query := TOF_Core.GenericValueFactory.FromIntReference(value := keys[2]);
position := _Dictionary.GetKeyPosition(key := keys[2]);
genericPosition := _Dictionary.GetGenericKeyPosition(key := query, releaseKey := FALSE);

Assert.ThatBool(
	actual := position >= 0 AND_THEN position < _Dictionary.Length,
	message := "Key 2 must have a valid current position"
).IsTrue();

Assert.ThatDInt(
	actual := genericPosition,
	message := "Both lookup forms must return the same position for key 2"
).ToBe(expected := position);

FOR i := 0 TO 6 DO
	found := _Dictionary.TryGetValueByKey(key := keys[i], value => value);

	IF i = 3 THEN
		Assert.ThatBool(
			actual := found AND_THEN value.AsString255() = copyReplacement,
			message := "SetCopy must replace the value of key 3"
		).IsTrue();
	ELSIF i = 5 THEN
		Assert.ThatBool(
			actual := found AND_THEN value.AsString255() = _ReplacementValue,
			message := "SetGeneric must replace the value of key 5"
		).IsTrue();
	ELSE
		Assert.ThatBool(
			actual := found AND_THEN value.AsString255() = values[i],
			message := TOF_Core.WideStrings.Concat255("Expected original value at key ", TO_WSTRING(i))
		).IsTrue();
	END_IF
END_FOR

found := _Dictionary.TryGetValueByGenericKey(key := query, releaseKey := FALSE, value => value);

Assert.ThatBool(
	actual := found AND_THEN value.AsString255() = 'String2',
	message := "Generic lookup must return the original value of key 2"
).IsTrue();

position := _Dictionary.GetKeyPosition(key := keys[3]);

IF position < 0 OR_ELSE position >= _Dictionary.Length THEN
	RecordFailure(message := "Updated key 3 must have a valid position");

	RETURN;
END_IF

pair REF= _Dictionary.GetKeyValuePairByIndex(index := position);

Assert.ThatBool(
	actual := __ISVALIDREF(pair) AND_THEN pair.Key.AsInt() = INT#3
		AND_THEN pair.Value.AsString255() = copyReplacement,
	message := "The indexed pair must match both the queried key and its updated value"
).IsTrue();
END_METHOD

(*!
<summary>Clears the fixture before the runner publishes the result.</summary>
<description>
Also runs after an unexpected exception interrupts the case.
</description>
*)
METHOD PROTECTED AfterTest
_Dictionary.Clear();
END_METHOD

//! <summary>Borrows the concrete class name. Callers must not modify it.</summary>
{attribute 'monitoring' := 'call'}
PROPERTY ClassName : REFERENCE TO STRING
GET
ClassName REF= _ClassName;
END_GET
END_PROPERTY

//! <summary>Borrows the compiler-initialized namespace name. Callers must not modify it.</summary>
{attribute 'monitoring' := 'call'}
PROPERTY NamespaceName : REFERENCE TO STRING
GET
NamespaceName REF= CurrentNamespace.Name;
END_GET
END_PROPERTY

//! <summary>Reports the concrete instance size in bytes.</summary>
{attribute 'monitoring' := 'call'}
PROPERTY SelfSize : ULINT
GET
SelfSize := XSIZEOF(THIS^);
END_GET
END_PROPERTY

END_FUNCTION_BLOCK

// ---- Tests/Collections/DictionaryRemoveTest.TcPOU
(*
SPDX-FileCopyrightText: c 2026 Oleksandr Tiutyk <trofimich@gmail.com>
SPDX-License-Identifier: MIT
License: https://opensource.org/license/mit
*)

(*!
<summary>Checks removal by current position and by both key forms.</summary>
<description>
Borrows one group-owned dictionary reserved for this case. Use from one task at a stable address.
Teardown clears entries owned by the dictionary before publication.
</description>
*)

{attribute 'no_assign'}
{attribute 'no_explicit_call' := 'do not call this function block directly'}
FUNCTION_BLOCK DictionaryRemoveTest EXTENDS TOF_Testing.SingleCycleTest
VAR_STAT
	{attribute 'hide'}
	_ClassName : STRING := __POUNAME();
END_VAR
VAR
	_Dictionary : TOF_Collections.IDictionary;
END_VAR

(*!
<summary>Clears the fixture before the runner publishes the result.</summary>
<description>
Also runs after an unexpected exception interrupts the case.
</description>
*)
METHOD PROTECTED AfterTest
_Dictionary.Clear();
END_METHOD

//! <summary>Borrows the concrete class name. Callers must not modify it.</summary>
{attribute 'monitoring' := 'call'}
PROPERTY ClassName : REFERENCE TO STRING
GET
ClassName REF= _ClassName;
END_GET
END_PROPERTY

(*!
<summary>Checks removal by current position and by both key forms.</summary>
*)
METHOD PROTECTED ExecuteTest
VAR
	keys : ARRAY [0..6] OF INT := [0, 1, 2, 3, 4, 5, 6];
	values : ARRAY [0..6] OF STRING :=
		['String0', 'String1', 'String2', 'String3', 'String4', 'String5', 'String6'];
	i : DINT;
	position : DINT;
	query : TOF_Core.GENERIC_VALUE;
	removed : BOOL;
END_VAR
FOR i := 6 TO 0 BY -1 DO
	_Dictionary.SetCopy(key := keys[i], value := values[i]);
END_FOR

_Dictionary.SetCopy(key := keys[3], value := values[3]);

position := _Dictionary.GetKeyPosition(key := keys[3]);

IF position < 0 OR_ELSE position >= _Dictionary.Length THEN
	RecordFailure(message := "Key 3 must have a valid position before removal");

	RETURN;
END_IF

_Dictionary.RemoveAt(index := position);

Assert.ThatBool(
	actual := _Dictionary.Length = 6 AND_THEN NOT _Dictionary.ContainsKey(key := keys[3]),
	message := "RemoveAt must remove only key 3"
).IsTrue();

_Dictionary.TryRemoveByKey(key := keys[2], removed => removed);

Assert.ThatBool(
	actual := removed AND_THEN _Dictionary.Length = 5 AND_THEN NOT _Dictionary.ContainsKey(key := keys[2]),
	message := "TryRemoveByKey must remove key 2 and report success"
).IsTrue();

query := TOF_Core.GenericValueFactory.FromIntReference(value := keys[1]);
_Dictionary.TryRemoveByGenericKey(key := query, releaseKey := FALSE, removed => removed);

Assert.ThatBool(
	actual := removed AND_THEN _Dictionary.Length = 4 AND_THEN NOT _Dictionary.ContainsKey(key := keys[1]),
	message := "TryRemoveByGenericKey must remove key 1 and report success"
).IsTrue();

_Dictionary.TryRemoveByGenericKey(key := query, releaseKey := FALSE, removed => removed);

Assert.ThatBool(
	actual := NOT removed AND_THEN _Dictionary.Length = 4,
	message := "A second removal of key 1 must leave the dictionary unchanged"
).IsTrue();

FOR i := 4 TO 6 DO
	Assert.ThatBool(
		actual := _Dictionary.ContainsKey(key := keys[i]),
		message := TOF_Core.WideStrings.Concat255("Removal must preserve key ", TO_WSTRING(i))
	).IsTrue();
END_FOR

Assert.ThatBool(
	actual := _Dictionary.ContainsKey(key := keys[0]),
	message := "Removal must preserve key 0"
).IsTrue();
END_METHOD

(*!
<summary>Binds the dictionary fixture for this case.</summary>
<description>
Stores a borrowed interface without invoking the fixture. The owning group keeps it alive and
reserves it for this case. TestElement initializes the name and parent.
</description>
<param name="name">Display name of this case.</param>
<param name="parent">Group that owns this case.</param>
<param name="dictionary">Required live dictionary reserved for this case.</param>
*)
METHOD FB_init : BOOL
VAR_INPUT
	bInitRetains: BOOL; // TRUE: the retain variables are initialized (reset warm / reset cold)
	bInCopyCode: BOOL; // TRUE: the instance will be copied to the copy code afterward (online change)
	name : WSTRING;
	parent : TOF_Testing.ITestElement;
	dictionary : TOF_Collections.IDictionary;
END_VAR
_Dictionary := dictionary;
FB_init := TRUE;
END_METHOD

//! <summary>Borrows the compiler-initialized namespace name. Callers must not modify it.</summary>
{attribute 'monitoring' := 'call'}
PROPERTY NamespaceName : REFERENCE TO STRING
GET
NamespaceName REF= CurrentNamespace.Name;
END_GET
END_PROPERTY

//! <summary>Reports the concrete instance size in bytes.</summary>
{attribute 'monitoring' := 'call'}
PROPERTY SelfSize : ULINT
GET
SelfSize := XSIZEOF(THIS^);
END_GET
END_PROPERTY

END_FUNCTION_BLOCK

// ---- Tests/Collections/DictionaryContainsTest.TcPOU
(*
SPDX-FileCopyrightText: c 2026 Oleksandr Tiutyk <trofimich@gmail.com>
SPDX-License-Identifier: MIT
License: https://opensource.org/license/mit
*)

(*!
<summary>Checks matching and missing keys with raw and borrowed generic queries.</summary>
<description>
Borrows one group-owned dictionary reserved for this case. Use from one task at a stable address.
Teardown clears entries owned by the dictionary before publication.
</description>
*)

{attribute 'no_assign'}
{attribute 'no_explicit_call' := 'do not call this function block directly'}
FUNCTION_BLOCK DictionaryContainsTest EXTENDS TOF_Testing.SingleCycleTest
VAR_STAT
	{attribute 'hide'}
	_ClassName : STRING := __POUNAME();
END_VAR
VAR
	_Dictionary : TOF_Collections.IDictionary;
END_VAR

(*!
<summary>Clears the fixture before the runner publishes the result.</summary>
<description>
Also runs after an unexpected exception interrupts the case.
</description>
*)
METHOD PROTECTED AfterTest
_Dictionary.Clear();
END_METHOD

//! <summary>Borrows the concrete class name. Callers must not modify it.</summary>
{attribute 'monitoring' := 'call'}
PROPERTY ClassName : REFERENCE TO STRING
GET
ClassName REF= _ClassName;
END_GET
END_PROPERTY

(*!
<summary>Checks matching and missing keys with raw and borrowed generic queries.</summary>
*)
METHOD PROTECTED ExecuteTest
VAR
	keys : ARRAY [0..6] OF INT := [0, 1, 2, 3, 4, 5, 6];
	values : ARRAY [0..6] OF STRING :=
		['String0', 'String1', 'String2', 'String3', 'String4', 'String5', 'String6'];
	i : DINT;
	missingKey : INT := 9;
	query : TOF_Core.GENERIC_VALUE;
END_VAR
FOR i := 6 TO 0 BY -1 DO
	_Dictionary.SetCopy(key := keys[i], value := values[i]);
END_FOR

_Dictionary.SetCopy(key := keys[3], value := values[3]);

Assert.ThatBool(
	actual := _Dictionary.ContainsKey(key := keys[3]),
	message := "ContainsKey must find the stored key"
).IsTrue();

Assert.ThatBool(
	actual := _Dictionary.ContainsKey(key := missingKey),
	message := "ContainsKey must reject an absent key"
).IsFalse();

query := TOF_Core.GenericValueFactory.FromIntReference(value := keys[3]);
Assert.ThatBool(
	actual := _Dictionary.ContainsGenericKey(key := query, releaseKey := FALSE),
	message := "ContainsGenericKey must find the stored key"
).IsTrue();

query := TOF_Core.GenericValueFactory.FromIntReference(value := missingKey);
Assert.ThatBool(
	actual := _Dictionary.ContainsGenericKey(key := query, releaseKey := FALSE),
	message := "ContainsGenericKey must reject an absent key"
).IsFalse();

Assert.ThatDInt(
	actual := _Dictionary.Length,
	message := "Lookup must preserve all seven entries"
).ToBe(expected := DINT#7);
END_METHOD

(*!
<summary>Binds the dictionary fixture for this case.</summary>
<description>
Stores a borrowed interface without invoking the fixture. The owning group keeps it alive and
reserves it for this case. TestElement initializes the name and parent.
</description>
<param name="name">Display name of this case.</param>
<param name="parent">Group that owns this case.</param>
<param name="dictionary">Required live dictionary reserved for this case.</param>
*)
METHOD FB_init : BOOL
VAR_INPUT
	bInitRetains: BOOL; // TRUE: the retain variables are initialized (reset warm / reset cold)
	bInCopyCode: BOOL; // TRUE: the instance will be copied to the copy code afterward (online change)
	name : WSTRING;
	parent : TOF_Testing.ITestElement;
	dictionary : TOF_Collections.IDictionary;
END_VAR
_Dictionary := dictionary;
FB_init := TRUE;
END_METHOD

//! <summary>Borrows the compiler-initialized namespace name. Callers must not modify it.</summary>
{attribute 'monitoring' := 'call'}
PROPERTY NamespaceName : REFERENCE TO STRING
GET
NamespaceName REF= CurrentNamespace.Name;
END_GET
END_PROPERTY

//! <summary>Reports the concrete instance size in bytes.</summary>
{attribute 'monitoring' := 'call'}
PROPERTY SelfSize : ULINT
GET
SelfSize := XSIZEOF(THIS^);
END_GET
END_PROPERTY

END_FUNCTION_BLOCK

// ---- Tests/Collections/Dynamic/DynamicDictionaryClearTest.TcPOU
(*
SPDX-FileCopyrightText: c 2026 Oleksandr Tiutyk <trofimich@gmail.com>
SPDX-License-Identifier: MIT
License: https://opensource.org/license/mit
*)

(*!
<summary>Checks clearing grown entries and rebuilding a usable index on reuse.</summary>
<description>
Owns a dynamic dictionary and copied pairs at a stable address. Run from one task.
Teardown releases remaining entries and dynamic storage.
</description>
*)

{attribute 'no_assign'}
{attribute 'no_explicit_call' := 'do not call this function block directly'}
FUNCTION_BLOCK DynamicDictionaryClearTest EXTENDS TOF_Testing.SingleCycleTest
VAR_STAT
	{attribute 'hide'}
	_ClassName : STRING := __POUNAME();
END_VAR
VAR
	_Dictionary : TOF_Collections.Dictionary<0>(keyValidator := 0, valueValidator := 0, keyEqualityComparer := 0);
END_VAR

(*!
<summary>Checks clearing grown entries and rebuilding a usable index on reuse.</summary>
*)
METHOD PROTECTED ExecuteTest
VAR
	keys : ARRAY [0..6] OF INT := [0, 1, 2, 3, 4, 5, 6];
	values : ARRAY [0..6] OF STRING :=
		['String0', 'String1', 'String2', 'String3', 'String4', 'String5', 'String6'];
	i : DINT;
	value : TOF_Core.GENERIC_VALUE;
	found : BOOL;
END_VAR
_Dictionary.DefaultDynamicAllocationElementCount := BYTE#2;

FOR i := 6 TO 0 BY -1 DO
	_Dictionary.SetCopy(key := keys[i], value := values[i]);
END_FOR

Assert.ThatBool(
	actual := _Dictionary.Length = 7 AND_THEN _Dictionary.Capacity = 8,
	message := "The clear fixture must start with grown capacity"
).IsTrue();

FOR i := 0 TO 6 DO
	found := _Dictionary.TryGetValueByKey(key := keys[i], value => value);

	Assert.ThatBool(
		actual := found AND_THEN value.AsString255() = values[i],
		message := TOF_Core.WideStrings.Concat255("Growth must preserve the pair at key ", TO_WSTRING(i))
	).IsTrue();
END_FOR

_Dictionary.Clear();

Assert.ThatBool(
	actual := _Dictionary.Empty AND_THEN _Dictionary.Length = 0 AND_THEN _Dictionary.Capacity = 0,
	message := "Clear must empty the dictionary and release capacity"
).IsTrue();

Assert.ThatBool(
	actual := _Dictionary.ContainsKey(key := keys[3]),
	message := "The cleared index must not find an old key"
).IsFalse();

_Dictionary.Clear();
_Dictionary.SetCopy(key := keys[3], value := values[6]);

found := _Dictionary.TryGetValueByKey(key := keys[3], value => value);

Assert.ThatBool(
	actual := found AND_THEN value.AsString255() = 'String6',
	message := "Reinsertion must make the new value visible"
).IsTrue();

Assert.ThatBool(
	actual := _Dictionary.Length = 1 AND_THEN _Dictionary.Capacity = 2,
	message := "Reinsertion must allocate only the initial capacity"
).IsTrue();
END_METHOD

(*!
<summary>Clears the fixture before the runner publishes the result.</summary>
<description>
Also runs after an unexpected exception interrupts the case.
</description>
*)
METHOD PROTECTED AfterTest
_Dictionary.Clear();
END_METHOD

//! <summary>Borrows the concrete class name. Callers must not modify it.</summary>
{attribute 'monitoring' := 'call'}
PROPERTY ClassName : REFERENCE TO STRING
GET
ClassName REF= _ClassName;
END_GET
END_PROPERTY

//! <summary>Borrows the compiler-initialized namespace name. Callers must not modify it.</summary>
{attribute 'monitoring' := 'call'}
PROPERTY NamespaceName : REFERENCE TO STRING
GET
NamespaceName REF= CurrentNamespace.Name;
END_GET
END_PROPERTY

//! <summary>Reports the concrete instance size in bytes.</summary>
{attribute 'monitoring' := 'call'}
PROPERTY SelfSize : ULINT
GET
SelfSize := XSIZEOF(THIS^);
END_GET
END_PROPERTY

END_FUNCTION_BLOCK

// ---- Tests/Collections/Static/StaticDictionaryTestGroup.TcPOU
(*
SPDX-FileCopyrightText: c 2026 Oleksandr Tiutyk <trofimich@gmail.com>
SPDX-License-Identifier: MIT
License: https://opensource.org/license/mit
*)

(*!
<summary>Groups fixed-capacity dictionary lookup, update, removal, clear and overflow cases.</summary>
<description>
Owns the child cases, their fixed registration array and the dictionaries borrowed by the common cases.
Each borrowed fixture is reserved for its case throughout the group lifetime. Use from one task at a stable address.
</description>
*)

{attribute 'no_assign'}
{attribute 'no_explicit_call' := 'do not call this function block directly'}
FUNCTION_BLOCK StaticDictionaryTestGroup EXTENDS TOF_Testing.TestGroup<5>
VAR_STAT
	{attribute 'hide'}
	_ClassName : STRING := __POUNAME();
END_VAR
VAR
	_SetAndGetDictionary : TOF_Collections.Dictionary<7>(keyValidator := 0, valueValidator := 0, keyEqualityComparer := 0);
	_RemoveDictionary : TOF_Collections.Dictionary<7>(keyValidator := 0, valueValidator := 0, keyEqualityComparer := 0);
	_ContainsDictionary : TOF_Collections.Dictionary<7>(keyValidator := 0, valueValidator := 0, keyEqualityComparer := 0);

	_SetAndGet : DictionarySetAndGetTest(name := "SetAndGet", parent := THIS^, dictionary := _SetAndGetDictionary);
	_Remove : DictionaryRemoveTest(name := "Remove", parent := THIS^, dictionary := _RemoveDictionary);
	_Contains : DictionaryContainsTest(name := "Contains", parent := THIS^, dictionary := _ContainsDictionary);
	_Clear : StaticDictionaryClearTest(name := "Clear", parent := THIS^);
	_Overflow : StaticDictionaryOverflowTest(name := "Overflow", parent := THIS^);

	_Children : ARRAY [0.._ChildCount - 1] OF TOF_Testing.ITestElement :=
	[
		_SetAndGet,
		_Remove,
		_Contains,
		_Clear,
		_Overflow
	];
END_VAR

//! <summary>Borrows the fixed child array. Callers must not modify it.</summary>
{attribute 'monitoring' := 'call'}
PROPERTY Children : REFERENCE TO ARRAY [0.._ChildCount - 1] OF TOF_Testing.ITestElement
GET
Children REF= _Children;
END_GET
END_PROPERTY

//! <summary>Borrows the concrete class name. Callers must not modify it.</summary>
{attribute 'monitoring' := 'call'}
PROPERTY ClassName : REFERENCE TO STRING
GET
ClassName REF= _ClassName;
END_GET
END_PROPERTY

//! <summary>Borrows the compiler-initialized namespace name. Callers must not modify it.</summary>
{attribute 'monitoring' := 'call'}
PROPERTY NamespaceName : REFERENCE TO STRING
GET
NamespaceName REF= CurrentNamespace.Name;
END_GET
END_PROPERTY

//! <summary>Reports the concrete instance size in bytes.</summary>
{attribute 'monitoring' := 'call'}
PROPERTY SelfSize : ULINT
GET
SelfSize := XSIZEOF(THIS^);
END_GET
END_PROPERTY

END_FUNCTION_BLOCK

// ---- Tests/Collections/Static/StaticDictionaryClearTest.TcPOU
(*
SPDX-FileCopyrightText: c 2026 Oleksandr Tiutyk <trofimich@gmail.com>
SPDX-License-Identifier: MIT
License: https://opensource.org/license/mit
*)

(*!
<summary>Checks clearing a full inline index and refilling its slots.</summary>
<description>
Owns a fixed-capacity dictionary and copied pairs at a stable address. Run from one task.
Teardown clears surviving entries before publication.
</description>
*)

{attribute 'no_assign'}
{attribute 'no_explicit_call' := 'do not call this function block directly'}
FUNCTION_BLOCK StaticDictionaryClearTest EXTENDS TOF_Testing.SingleCycleTest
VAR_STAT
	{attribute 'hide'}
	_ClassName : STRING := __POUNAME();
END_VAR
VAR
	_Dictionary : TOF_Collections.Dictionary<7>(keyValidator := 0, valueValidator := 0, keyEqualityComparer := 0);
END_VAR

(*!
<summary>Checks clearing a full inline index and refilling its slots.</summary>
*)
METHOD PROTECTED ExecuteTest
VAR
	keys : ARRAY [0..6] OF INT := [0, 1, 2, 3, 4, 5, 6];
	values : ARRAY [0..6] OF STRING :=
		['String0', 'String1', 'String2', 'String3', 'String4', 'String5', 'String6'];
	i : DINT;
	value : TOF_Core.GENERIC_VALUE;
	found : BOOL;
END_VAR
FOR i := 6 TO 0 BY -1 DO
	_Dictionary.SetCopy(key := keys[i], value := values[i]);
END_FOR

Assert.ThatBool(
	actual := _Dictionary.Full AND_THEN _Dictionary.Length = 7,
	message := "The clear fixture must start full"
).IsTrue();

_Dictionary.Clear();

Assert.ThatBool(
	actual := _Dictionary.Empty AND_THEN _Dictionary.Length = 0 AND_THEN NOT _Dictionary.Full,
	message := "Clearing a full dictionary must make every slot available"
).IsTrue();

Assert.ThatDInt(
	actual := _Dictionary.Capacity,
	message := "Clearing must preserve inline capacity"
).ToBe(expected := DINT#7);

FOR i := 0 TO 6 DO
	Assert.ThatBool(
		actual := _Dictionary.ContainsKey(key := keys[i]),
		message := TOF_Core.WideStrings.Concat255("Clear must hide old key ", TO_WSTRING(i))
	).IsFalse();
END_FOR

FOR i := 0 TO 6 DO
	_Dictionary.SetCopy(key := keys[i], value := values[6 - i]);
END_FOR

Assert.ThatBool(
	actual := _Dictionary.Full AND_THEN _Dictionary.Length = 7,
	message := "Refilling must reuse all seven slots"
).IsTrue();

FOR i := 0 TO 6 DO
	found := _Dictionary.TryGetValueByKey(key := keys[i], value => value);

	Assert.ThatBool(
		actual := found AND_THEN value.AsString255() = values[6 - i],
		message := TOF_Core.WideStrings.Concat255("Refill must return the new value at key ", TO_WSTRING(i))
	).IsTrue();
END_FOR
END_METHOD

(*!
<summary>Clears the fixture before the runner publishes the result.</summary>
<description>
Also runs after an unexpected exception interrupts the case.
</description>
*)
METHOD PROTECTED AfterTest
_Dictionary.Clear();
END_METHOD

//! <summary>Borrows the concrete class name. Callers must not modify it.</summary>
{attribute 'monitoring' := 'call'}
PROPERTY ClassName : REFERENCE TO STRING
GET
ClassName REF= _ClassName;
END_GET
END_PROPERTY

//! <summary>Borrows the compiler-initialized namespace name. Callers must not modify it.</summary>
{attribute 'monitoring' := 'call'}
PROPERTY NamespaceName : REFERENCE TO STRING
GET
NamespaceName REF= CurrentNamespace.Name;
END_GET
END_PROPERTY

//! <summary>Reports the concrete instance size in bytes.</summary>
{attribute 'monitoring' := 'call'}
PROPERTY SelfSize : ULINT
GET
SelfSize := XSIZEOF(THIS^);
END_GET
END_PROPERTY

END_FUNCTION_BLOCK

// ---- Tests/Collections/Static/StaticDictionaryOverflowTest.TcPOU
(*
SPDX-FileCopyrightText: c 2026 Oleksandr Tiutyk <trofimich@gmail.com>
SPDX-License-Identifier: MIT
License: https://opensource.org/license/mit
*)

(*!
<summary>Checks rejection of a new key at capacity and reuse after removal.</summary>
<description>
Owns a fixed-capacity dictionary and copied pairs at a stable address. Run from one task.
Teardown clears surviving entries before publication.
</description>
*)

{attribute 'no_assign'}
{attribute 'no_explicit_call' := 'do not call this function block directly'}
FUNCTION_BLOCK StaticDictionaryOverflowTest EXTENDS TOF_Testing.SingleCycleTest
VAR_STAT
	{attribute 'hide'}
	_ClassName : STRING := __POUNAME();
END_VAR
VAR
	_Dictionary : TOF_Collections.Dictionary<7>(keyValidator := 0, valueValidator := 0, keyEqualityComparer := 0);
END_VAR

(*!
<summary>Checks rejection of a new key at capacity and reuse after removal.</summary>
*)
METHOD PROTECTED ExecuteTest
VAR
	keys : ARRAY [0..6] OF INT := [0, 1, 2, 3, 4, 5, 6];
	values : ARRAY [0..6] OF STRING :=
		['String0', 'String1', 'String2', 'String3', 'String4', 'String5', 'String6'];
	i : DINT;
	newKey : INT := 7;
	newValue : STRING := 'String7';
	found : BOOL;
	removed : BOOL;
	value : TOF_Core.GENERIC_VALUE;

	exceptionCode : __SYSTEM.ExceptionCode;
	caught : TOF_Core.IException;
	fullException : TOF_Core.IStaticCollectionFullException;
END_VAR
FOR i := 6 TO 0 BY -1 DO
	_Dictionary.SetCopy(key := keys[i], value := values[i]);
END_FOR

Assert.ThatBool(
	actual := _Dictionary.Full AND_THEN _Dictionary.Length = 7,
	message := "The overflow fixture must start full"
).IsTrue();

__TRY
	_Dictionary.SetCopy(key := newKey, value := newValue);
__CATCH(exceptionCode)
	caught := TOF_Core.ExceptionManager.GetLastException(
		exceptionCode := exceptionCode,
		catchPointNamespaceName := NamespaceName,
		catchPointPOUName := __POUNAME(),
		catchPointPosition := __POSITION()
	);
__ENDTRY

Assert.ThatBool(
	actual := __QUERYINTERFACE(caught, fullException),
	message := "Adding a new key at capacity must raise StaticCollectionFullException"
).IsTrue();

Assert.ThatBool(
	actual := _Dictionary.Full AND_THEN _Dictionary.Length = 7 AND_THEN _Dictionary.Capacity = 7,
	message := "Rejected insertion must preserve full length and capacity"
).IsTrue();

Assert.ThatBool(
	actual := _Dictionary.ContainsKey(key := newKey),
	message := "The rejected key must remain absent"
).IsFalse();

FOR i := 0 TO 6 DO
	found := _Dictionary.TryGetValueByKey(key := keys[i], value => value);

	Assert.ThatBool(
		actual := found AND_THEN value.AsString255() = values[i],
		message := TOF_Core.WideStrings.Concat255("Overflow must preserve the original pair at key ", TO_WSTRING(i))
	).IsTrue();
END_FOR

_Dictionary.TryRemoveByKey(key := keys[3], removed => removed);

Assert.ThatBool(
	actual := removed,
	message := "Removing an existing key must free a slot"
).IsTrue();

_Dictionary.SetCopy(key := newKey, value := newValue);
found := _Dictionary.TryGetValueByKey(key := newKey, value => value);

Assert.ThatBool(
	actual := _Dictionary.Full AND_THEN found AND_THEN value.AsString255() = newValue,
	message := "Reusing a slot must make the new pair visible"
).IsTrue();

Assert.ThatBool(
	actual := _Dictionary.ContainsKey(key := keys[3]),
	message := "Reusing the slot must keep the removed key absent"
).IsFalse();
END_METHOD

(*!
<summary>Clears the fixture before the runner publishes the result.</summary>
<description>
Also runs after an unexpected exception interrupts the case.
</description>
*)
METHOD PROTECTED AfterTest
_Dictionary.Clear();
END_METHOD

//! <summary>Borrows the concrete class name. Callers must not modify it.</summary>
{attribute 'monitoring' := 'call'}
PROPERTY ClassName : REFERENCE TO STRING
GET
ClassName REF= _ClassName;
END_GET
END_PROPERTY

//! <summary>Borrows the compiler-initialized namespace name. Callers must not modify it.</summary>
{attribute 'monitoring' := 'call'}
PROPERTY NamespaceName : REFERENCE TO STRING
GET
NamespaceName REF= CurrentNamespace.Name;
END_GET
END_PROPERTY

//! <summary>Reports the concrete instance size in bytes.</summary>
{attribute 'monitoring' := 'call'}
PROPERTY SelfSize : ULINT
GET
SelfSize := XSIZEOF(THIS^);
END_GET
END_PROPERTY

END_FUNCTION_BLOCK

// ---- Tests/Collections/Dynamic/DynamicUniqueDataSetTestGroup.TcPOU
(*
SPDX-FileCopyrightText: c 2026 Oleksandr Tiutyk <trofimich@gmail.com>
SPDX-License-Identifier: MIT
License: https://opensource.org/license/mit
*)

(*!
<summary>Groups dynamic set lookup, duplicate updates, removal and clear cases.</summary>
<description>
Owns the child cases, their fixed registration array and the sets borrowed by the common cases.
Each borrowed fixture is reserved for its case throughout the group lifetime. Use from one task at a stable address.
</description>
*)

{attribute 'no_assign'}
{attribute 'no_explicit_call' := 'do not call this function block directly'}
FUNCTION_BLOCK DynamicUniqueDataSetTestGroup EXTENDS TOF_Testing.TestGroup<4>
VAR_STAT
	{attribute 'hide'}
	_ClassName : STRING := __POUNAME();
END_VAR
VAR
	_SetAndGetSet : TOF_Collections.UniqueDataSet<0>(valueValidator := 0, valueEqualityComparer := 0);
	_RemoveSet : TOF_Collections.UniqueDataSet<0>(valueValidator := 0, valueEqualityComparer := 0);
	_ContainsSet : TOF_Collections.UniqueDataSet<0>(valueValidator := 0, valueEqualityComparer := 0);

	_SetAndGet : UniqueDataSetSetAndGetTest(name := "SetAndGet", parent := THIS^, dataSet := _SetAndGetSet);
	_Remove : UniqueDataSetRemoveTest(name := "Remove", parent := THIS^, dataSet := _RemoveSet);
	_Contains : UniqueDataSetContainsTest(name := "Contains", parent := THIS^, dataSet := _ContainsSet);
	_Clear : DynamicUniqueDataSetClearTest(name := "Clear", parent := THIS^);

	_Children : ARRAY [0.._ChildCount - 1] OF TOF_Testing.ITestElement :=
	[
		_SetAndGet,
		_Remove,
		_Contains,
		_Clear
	];
END_VAR

//! <summary>Borrows the fixed child array. Callers must not modify it.</summary>
{attribute 'monitoring' := 'call'}
PROPERTY Children : REFERENCE TO ARRAY [0.._ChildCount - 1] OF TOF_Testing.ITestElement
GET
Children REF= _Children;
END_GET
END_PROPERTY

//! <summary>Borrows the concrete class name. Callers must not modify it.</summary>
{attribute 'monitoring' := 'call'}
PROPERTY ClassName : REFERENCE TO STRING
GET
ClassName REF= _ClassName;
END_GET
END_PROPERTY

//! <summary>Borrows the compiler-initialized namespace name. Callers must not modify it.</summary>
{attribute 'monitoring' := 'call'}
PROPERTY NamespaceName : REFERENCE TO STRING
GET
NamespaceName REF= CurrentNamespace.Name;
END_GET
END_PROPERTY

//! <summary>Reports the concrete instance size in bytes.</summary>
{attribute 'monitoring' := 'call'}
PROPERTY SelfSize : ULINT
GET
SelfSize := XSIZEOF(THIS^);
END_GET
END_PROPERTY

END_FUNCTION_BLOCK

// ---- Tests/Collections/UniqueDataSetSetAndGetTest.TcPOU
(*
SPDX-FileCopyrightText: c 2026 Oleksandr Tiutyk <trofimich@gmail.com>
SPDX-License-Identifier: MIT
License: https://opensource.org/license/mit
*)

(*!
<summary>Checks copy and generic insertion, duplicate updates and indexed values.</summary>
<description>
Borrows one group-owned set reserved for this case. Use from one task at a stable address.
Teardown clears the set and releases its owned entries before publication.
</description>
*)

{attribute 'no_assign'}
{attribute 'no_explicit_call' := 'do not call this function block directly'}
FUNCTION_BLOCK UniqueDataSetSetAndGetTest EXTENDS TOF_Testing.SingleCycleTest
VAR_STAT
	{attribute 'hide'}
	_ClassName : STRING := __POUNAME();
END_VAR
VAR
	_Set : TOF_Collections.IUniqueDataSet;
	_GenericValues : ARRAY [0..2] OF STRING := ['String3', 'String5', 'String6'];
END_VAR

(*!
<summary>Binds the unique set fixture for this case.</summary>
<description>
Stores a borrowed interface without invoking the fixture. The owning group keeps it alive and
reserves it for this case. TestElement initializes the name and parent.
</description>
<param name="name">Display name of this case.</param>
<param name="parent">Group that owns this case.</param>
<param name="dataSet">Required live unique set reserved for this case.</param>
*)
METHOD FB_init : BOOL
VAR_INPUT
	bInitRetains: BOOL; // TRUE: the retain variables are initialized (reset warm / reset cold)
	bInCopyCode: BOOL; // TRUE: the instance will be copied to the copy code afterward (online change)
	name : WSTRING;
	parent : TOF_Testing.ITestElement;
	dataSet : TOF_Collections.IUniqueDataSet;
END_VAR
_Set := dataSet;
FB_init := TRUE;
END_METHOD

(*!
<summary>Checks copy and generic insertion, duplicate updates and indexed values.</summary>
*)
METHOD PROTECTED ExecuteTest
VAR
	values : ARRAY [0..6] OF STRING :=
		['String0', 'String1', 'String2', 'String3', 'String4', 'String5', 'String6'];
	i : DINT;
	position : DINT;
	genericPosition : DINT;
	insertedPosition : DINT;

	query : TOF_Core.GENERIC_VALUE;
	entry : REFERENCE TO TOF_Core.GENERIC_VALUE;
	diagnostic : TOF_Core.ERROR_MESSAGE;
END_VAR
FOR i := 5 TO 0 BY -1 DO
	_Set.SetCopy(value := values[i]);
END_FOR

query := TOF_Core.GenericValueFactory.FromStringReference(value := _GenericValues[2]);
_Set.SetGeneric(value := query, index => insertedPosition);

Assert.ThatDInt(
	actual := _Set.Length,
	message := "SetGeneric must insert a new seventh value"
).ToBe(expected := DINT#7);

Assert.ThatDInt(
	actual := _Set.GetValuePosition(value := values[6]),
	message := "SetGeneric must report the position of the inserted value"
).ToBe(expected := insertedPosition);

_Set.SetCopy(value := values[3]);

FOR i := 0 TO 1 DO
	query := TOF_Core.GenericValueFactory.FromStringReference(value := _GenericValues[i]);
	_Set.SetGeneric(value := query);
END_FOR

Assert.ThatDInt(
	actual := _Set.Length,
	message := "Duplicate updates must preserve length"
).ToBe(expected := DINT#7);

query := TOF_Core.GenericValueFactory.FromStringReference(value := values[2]);
position := _Set.GetValuePosition(value := values[2]);
genericPosition := _Set.GetGenericValuePosition(value := query, releaseValue := FALSE);

Assert.ThatBool(
	actual := position >= 0 AND_THEN position < _Set.Length,
	message := "String2 must have a valid current position"
).IsTrue();

Assert.ThatDInt(
	actual := genericPosition,
	message := "Both lookup forms must return the same position for String2"
).ToBe(expected := position);

FOR i := 0 TO 6 DO
	position := _Set.GetValuePosition(value := values[i]);

	IF position < 0 OR_ELSE position >= _Set.Length THEN
		diagnostic := TOF_Core.WideStrings.Concat255("Missing value at source offset ", TO_WSTRING(i));
		RecordFailure(message := diagnostic);

		RETURN;
	END_IF

	entry REF= _Set.GetByIndex(index := position);
	Assert.ThatBool(
		actual := __ISVALIDREF(entry) AND_THEN entry.AsString255() = values[i],
		message := TOF_Core.WideStrings.Concat255("Indexed lookup must match the value at offset ", TO_WSTRING(i))
	).IsTrue();
END_FOR
END_METHOD

(*!
<summary>Clears the fixture before the runner publishes the result.</summary>
<description>
Also runs after an unexpected exception interrupts the case.
</description>
*)
METHOD PROTECTED AfterTest
_Set.Clear();
END_METHOD

//! <summary>Borrows the concrete class name. Callers must not modify it.</summary>
{attribute 'monitoring' := 'call'}
PROPERTY ClassName : REFERENCE TO STRING
GET
ClassName REF= _ClassName;
END_GET
END_PROPERTY

//! <summary>Borrows the compiler-initialized namespace name. Callers must not modify it.</summary>
{attribute 'monitoring' := 'call'}
PROPERTY NamespaceName : REFERENCE TO STRING
GET
NamespaceName REF= CurrentNamespace.Name;
END_GET
END_PROPERTY

//! <summary>Reports the concrete instance size in bytes.</summary>
{attribute 'monitoring' := 'call'}
PROPERTY SelfSize : ULINT
GET
SelfSize := XSIZEOF(THIS^);
END_GET
END_PROPERTY

END_FUNCTION_BLOCK

// ---- Tests/Collections/UniqueDataSetRemoveTest.TcPOU
(*
SPDX-FileCopyrightText: c 2026 Oleksandr Tiutyk <trofimich@gmail.com>
SPDX-License-Identifier: MIT
License: https://opensource.org/license/mit
*)

(*!
<summary>Checks positional, raw and generic removal with stable membership afterward.</summary>
<description>
Borrows one group-owned set reserved for this case. Use from one task at a stable address.
Teardown clears the set and releases its owned entries before publication.
</description>
*)

{attribute 'no_assign'}
{attribute 'no_explicit_call' := 'do not call this function block directly'}
FUNCTION_BLOCK UniqueDataSetRemoveTest EXTENDS TOF_Testing.SingleCycleTest
VAR_STAT
	{attribute 'hide'}
	_ClassName : STRING := __POUNAME();
END_VAR
VAR
	_Set : TOF_Collections.IUniqueDataSet;
END_VAR

(*!
<summary>Clears the fixture before the runner publishes the result.</summary>
<description>
Also runs after an unexpected exception interrupts the case.
</description>
*)
METHOD PROTECTED AfterTest
_Set.Clear();
END_METHOD

//! <summary>Borrows the concrete class name. Callers must not modify it.</summary>
{attribute 'monitoring' := 'call'}
PROPERTY ClassName : REFERENCE TO STRING
GET
ClassName REF= _ClassName;
END_GET
END_PROPERTY

(*!
<summary>Checks positional, raw and generic removal with stable membership afterward.</summary>
*)
METHOD PROTECTED ExecuteTest
VAR
	values : ARRAY [0..6] OF STRING :=
		['String0', 'String1', 'String2', 'String3', 'String4', 'String5', 'String6'];
	i : DINT;
	position : DINT;
	removed : BOOL;
	query : TOF_Core.GENERIC_VALUE;
END_VAR
FOR i := 6 TO 0 BY -1 DO
	_Set.SetCopy(value := values[i]);
END_FOR

position := _Set.GetValuePosition(value := values[3]);

IF position < 0 OR_ELSE position >= _Set.Length THEN
	RecordFailure(message := "String3 must have a valid position before removal");

	RETURN;
END_IF

_Set.RemoveAt(index := position);

Assert.ThatBool(
	actual := _Set.Length = 6 AND_THEN NOT _Set.Contains(value := values[3]),
	message := "RemoveAt must remove String3 from the set"
).IsTrue();

_Set.TryRemove(value := values[2], removed => removed);

Assert.ThatBool(
	actual := removed AND_THEN _Set.Length = 5 AND_THEN NOT _Set.Contains(value := values[2]),
	message := "TryRemove must remove String2 and report success"
).IsTrue();

query := TOF_Core.GenericValueFactory.FromStringReference(value := values[1]);
_Set.TryRemoveGeneric(value := query, releaseValue := FALSE, removed => removed);

Assert.ThatBool(
	actual := removed AND_THEN _Set.Length = 4 AND_THEN NOT _Set.Contains(value := values[1]),
	message := "TryRemoveGeneric must remove String1 and report success"
).IsTrue();

_Set.TryRemoveGeneric(value := query, releaseValue := FALSE, removed => removed);

Assert.ThatBool(
	actual := NOT removed AND_THEN _Set.Length = 4,
	message := "Repeating removal of String1 must leave the set unchanged"
).IsTrue();

FOR i := 4 TO 6 DO
	Assert.ThatBool(
		actual := _Set.Contains(value := values[i]),
		message := TOF_Core.WideStrings.Concat255("Removal must preserve the value at offset ", TO_WSTRING(i))
	).IsTrue();
END_FOR

Assert.ThatBool(
	actual := _Set.Contains(value := values[0]),
	message := "Removal must preserve String0"
).IsTrue();
END_METHOD

(*!
<summary>Binds the unique set fixture for this case.</summary>
<description>
Stores a borrowed interface without invoking the fixture. The owning group keeps it alive and
reserves it for this case. TestElement initializes the name and parent.
</description>
<param name="name">Display name of this case.</param>
<param name="parent">Group that owns this case.</param>
<param name="dataSet">Required live unique set reserved for this case.</param>
*)
METHOD FB_init : BOOL
VAR_INPUT
	bInitRetains: BOOL; // TRUE: the retain variables are initialized (reset warm / reset cold)
	bInCopyCode: BOOL; // TRUE: the instance will be copied to the copy code afterward (online change)
	name : WSTRING;
	parent : TOF_Testing.ITestElement;
	dataSet : TOF_Collections.IUniqueDataSet;
END_VAR
_Set := dataSet;
FB_init := TRUE;
END_METHOD

//! <summary>Borrows the compiler-initialized namespace name. Callers must not modify it.</summary>
{attribute 'monitoring' := 'call'}
PROPERTY NamespaceName : REFERENCE TO STRING
GET
NamespaceName REF= CurrentNamespace.Name;
END_GET
END_PROPERTY

//! <summary>Reports the concrete instance size in bytes.</summary>
{attribute 'monitoring' := 'call'}
PROPERTY SelfSize : ULINT
GET
SelfSize := XSIZEOF(THIS^);
END_GET
END_PROPERTY

END_FUNCTION_BLOCK

// ---- Tests/Collections/UniqueDataSetContainsTest.TcPOU
(*
SPDX-FileCopyrightText: c 2026 Oleksandr Tiutyk <trofimich@gmail.com>
SPDX-License-Identifier: MIT
License: https://opensource.org/license/mit
*)

(*!
<summary>Checks stable membership for raw and generic matching and missing values.</summary>
<description>
Borrows one group-owned set reserved for this case. Use from one task at a stable address.
Teardown clears the set and releases its owned entries before publication.
</description>
*)

{attribute 'no_assign'}
{attribute 'no_explicit_call' := 'do not call this function block directly'}
FUNCTION_BLOCK UniqueDataSetContainsTest EXTENDS TOF_Testing.SingleCycleTest
VAR_STAT
	{attribute 'hide'}
	_ClassName : STRING := __POUNAME();
END_VAR
VAR
	_Set : TOF_Collections.IUniqueDataSet;
END_VAR

(*!
<summary>Clears the fixture before the runner publishes the result.</summary>
<description>
Also runs after an unexpected exception interrupts the case.
</description>
*)
METHOD PROTECTED AfterTest
_Set.Clear();
END_METHOD

//! <summary>Borrows the concrete class name. Callers must not modify it.</summary>
{attribute 'monitoring' := 'call'}
PROPERTY ClassName : REFERENCE TO STRING
GET
ClassName REF= _ClassName;
END_GET
END_PROPERTY

(*!
<summary>Checks stable membership for raw and generic matching and missing values.</summary>
*)
METHOD PROTECTED ExecuteTest
VAR
	values : ARRAY [0..6] OF STRING :=
		['String0', 'String1', 'String2', 'String3', 'String4', 'String5', 'String6'];
	i : DINT;
	missingValue : STRING := 'String9';
	query : TOF_Core.GENERIC_VALUE;
END_VAR
FOR i := 6 TO 0 BY -1 DO
	_Set.SetCopy(value := values[i]);
END_FOR

Assert.ThatBool(
	actual := _Set.Contains(value := values[3]),
	message := "Contains must find a stored value"
).IsTrue();

Assert.ThatBool(
	actual := _Set.Contains(value := missingValue),
	message := "Contains must reject an absent value"
).IsFalse();

query := TOF_Core.GenericValueFactory.FromStringReference(value := values[3]);
Assert.ThatBool(
	actual := _Set.ContainsGeneric(value := query, releaseValue := FALSE),
	message := "ContainsGeneric must find a stored value"
).IsTrue();

query := TOF_Core.GenericValueFactory.FromStringReference(value := missingValue);
Assert.ThatBool(
	actual := _Set.ContainsGeneric(value := query, releaseValue := FALSE),
	message := "ContainsGeneric must reject an absent value"
).IsFalse();

Assert.ThatDInt(
	actual := _Set.Length,
	message := "Lookup must preserve all seven entries"
).ToBe(expected := DINT#7);
END_METHOD

(*!
<summary>Binds the unique set fixture for this case.</summary>
<description>
Stores a borrowed interface without invoking the fixture. The owning group keeps it alive and
reserves it for this case. TestElement initializes the name and parent.
</description>
<param name="name">Display name of this case.</param>
<param name="parent">Group that owns this case.</param>
<param name="dataSet">Required live unique set reserved for this case.</param>
*)
METHOD FB_init : BOOL
VAR_INPUT
	bInitRetains: BOOL; // TRUE: the retain variables are initialized (reset warm / reset cold)
	bInCopyCode: BOOL; // TRUE: the instance will be copied to the copy code afterward (online change)
	name : WSTRING;
	parent : TOF_Testing.ITestElement;
	dataSet : TOF_Collections.IUniqueDataSet;
END_VAR
_Set := dataSet;
FB_init := TRUE;
END_METHOD

//! <summary>Borrows the compiler-initialized namespace name. Callers must not modify it.</summary>
{attribute 'monitoring' := 'call'}
PROPERTY NamespaceName : REFERENCE TO STRING
GET
NamespaceName REF= CurrentNamespace.Name;
END_GET
END_PROPERTY

//! <summary>Reports the concrete instance size in bytes.</summary>
{attribute 'monitoring' := 'call'}
PROPERTY SelfSize : ULINT
GET
SelfSize := XSIZEOF(THIS^);
END_GET
END_PROPERTY

END_FUNCTION_BLOCK

// ---- Tests/Collections/Dynamic/DynamicUniqueDataSetClearTest.TcPOU
(*
SPDX-FileCopyrightText: c 2026 Oleksandr Tiutyk <trofimich@gmail.com>
SPDX-License-Identifier: MIT
License: https://opensource.org/license/mit
*)

(*!
<summary>Checks clearing grown storage and rebuilding membership on reuse.</summary>
<description>
Owns a dynamic set and copied values at a stable address. Run from one task.
Teardown releases remaining entries and dynamic storage.
</description>
*)

{attribute 'no_assign'}
{attribute 'no_explicit_call' := 'do not call this function block directly'}
FUNCTION_BLOCK DynamicUniqueDataSetClearTest EXTENDS TOF_Testing.SingleCycleTest
VAR_STAT
	{attribute 'hide'}
	_ClassName : STRING := __POUNAME();
END_VAR
VAR
	_Set : TOF_Collections.UniqueDataSet<0>(valueValidator := 0, valueEqualityComparer := 0);
END_VAR

(*!
<summary>Checks clearing grown storage and rebuilding membership on reuse.</summary>
*)
METHOD PROTECTED ExecuteTest
VAR
	values : ARRAY [0..6] OF STRING :=
		['String0', 'String1', 'String2', 'String3', 'String4', 'String5', 'String6'];
	i : DINT;
	freshValue : STRING := 'String9';
END_VAR
_Set.DefaultDynamicAllocationElementCount := BYTE#2;

FOR i := 6 TO 0 BY -1 DO
	_Set.SetCopy(value := values[i]);
END_FOR

Assert.ThatBool(
	actual := _Set.Length = 7 AND_THEN _Set.Capacity = 8,
	message := "The clear fixture must start with grown capacity"
).IsTrue();

FOR i := 0 TO 6 DO
	Assert.ThatBool(
		actual := _Set.Contains(value := values[i]),
		message := TOF_Core.WideStrings.Concat255("Growth must preserve the value at offset ", TO_WSTRING(i))
	).IsTrue();
END_FOR

_Set.Clear();

Assert.ThatBool(
	actual := _Set.Empty AND_THEN _Set.Length = 0 AND_THEN _Set.Capacity = 0,
	message := "Clear must empty the set and release capacity"
).IsTrue();

Assert.ThatBool(
	actual := _Set.Contains(value := values[3]),
	message := "The cleared index must not find an old member"
).IsFalse();

_Set.Clear();
_Set.SetCopy(value := freshValue);

Assert.ThatBool(
	actual := _Set.Contains(value := freshValue),
	message := "Reuse must index the newly inserted member"
).IsTrue();

Assert.ThatBool(
	actual := _Set.Contains(value := values[3]),
	message := "Reuse must keep old membership absent"
).IsFalse();

Assert.ThatBool(
	actual := _Set.Length = 1 AND_THEN _Set.Capacity = 2,
	message := "Reuse must allocate only the initial capacity"
).IsTrue();
END_METHOD

(*!
<summary>Clears the fixture before the runner publishes the result.</summary>
<description>
Also runs after an unexpected exception interrupts the case.
</description>
*)
METHOD PROTECTED AfterTest
_Set.Clear();
END_METHOD

//! <summary>Borrows the concrete class name. Callers must not modify it.</summary>
{attribute 'monitoring' := 'call'}
PROPERTY ClassName : REFERENCE TO STRING
GET
ClassName REF= _ClassName;
END_GET
END_PROPERTY

//! <summary>Borrows the compiler-initialized namespace name. Callers must not modify it.</summary>
{attribute 'monitoring' := 'call'}
PROPERTY NamespaceName : REFERENCE TO STRING
GET
NamespaceName REF= CurrentNamespace.Name;
END_GET
END_PROPERTY

//! <summary>Reports the concrete instance size in bytes.</summary>
{attribute 'monitoring' := 'call'}
PROPERTY SelfSize : ULINT
GET
SelfSize := XSIZEOF(THIS^);
END_GET
END_PROPERTY

END_FUNCTION_BLOCK

// ---- Tests/Collections/Static/StaticUniqueDataSetTestGroup.TcPOU
(*
SPDX-FileCopyrightText: c 2026 Oleksandr Tiutyk <trofimich@gmail.com>
SPDX-License-Identifier: MIT
License: https://opensource.org/license/mit
*)

(*!
<summary>Groups fixed-capacity set lookup, duplicate updates, removal, clear and overflow cases.</summary>
<description>
Owns the child cases, their fixed registration array and the sets borrowed by the common cases.
Each borrowed fixture is reserved for its case throughout the group lifetime. Use from one task at a stable address.
</description>
*)

{attribute 'no_assign'}
{attribute 'no_explicit_call' := 'do not call this function block directly'}
FUNCTION_BLOCK StaticUniqueDataSetTestGroup EXTENDS TOF_Testing.TestGroup<5>
VAR_STAT
	{attribute 'hide'}
	_ClassName : STRING := __POUNAME();
END_VAR
VAR
	_SetAndGetSet : TOF_Collections.UniqueDataSet<7>(valueValidator := 0, valueEqualityComparer := 0);
	_RemoveSet : TOF_Collections.UniqueDataSet<7>(valueValidator := 0, valueEqualityComparer := 0);
	_ContainsSet : TOF_Collections.UniqueDataSet<7>(valueValidator := 0, valueEqualityComparer := 0);

	_SetAndGet : UniqueDataSetSetAndGetTest(name := "SetAndGet", parent := THIS^, dataSet := _SetAndGetSet);
	_Remove : UniqueDataSetRemoveTest(name := "Remove", parent := THIS^, dataSet := _RemoveSet);
	_Contains : UniqueDataSetContainsTest(name := "Contains", parent := THIS^, dataSet := _ContainsSet);
	_Clear : StaticUniqueDataSetClearTest(name := "Clear", parent := THIS^);
	_Overflow : StaticUniqueDataSetOverflowTest(name := "Overflow", parent := THIS^);

	_Children : ARRAY [0.._ChildCount - 1] OF TOF_Testing.ITestElement :=
	[
		_SetAndGet,
		_Remove,
		_Contains,
		_Clear,
		_Overflow
	];
END_VAR

//! <summary>Borrows the fixed child array. Callers must not modify it.</summary>
{attribute 'monitoring' := 'call'}
PROPERTY Children : REFERENCE TO ARRAY [0.._ChildCount - 1] OF TOF_Testing.ITestElement
GET
Children REF= _Children;
END_GET
END_PROPERTY

//! <summary>Borrows the concrete class name. Callers must not modify it.</summary>
{attribute 'monitoring' := 'call'}
PROPERTY ClassName : REFERENCE TO STRING
GET
ClassName REF= _ClassName;
END_GET
END_PROPERTY

//! <summary>Borrows the compiler-initialized namespace name. Callers must not modify it.</summary>
{attribute 'monitoring' := 'call'}
PROPERTY NamespaceName : REFERENCE TO STRING
GET
NamespaceName REF= CurrentNamespace.Name;
END_GET
END_PROPERTY

//! <summary>Reports the concrete instance size in bytes.</summary>
{attribute 'monitoring' := 'call'}
PROPERTY SelfSize : ULINT
GET
SelfSize := XSIZEOF(THIS^);
END_GET
END_PROPERTY

END_FUNCTION_BLOCK

// ---- Tests/Collections/Static/StaticUniqueDataSetClearTest.TcPOU
(*
SPDX-FileCopyrightText: c 2026 Oleksandr Tiutyk <trofimich@gmail.com>
SPDX-License-Identifier: MIT
License: https://opensource.org/license/mit
*)

(*!
<summary>Checks clearing a full inline index and refilling with distinct values.</summary>
<description>
Owns a fixed-capacity set and copied values at a stable address. Run from one task.
Teardown clears surviving entries before publication.
</description>
*)

{attribute 'no_assign'}
{attribute 'no_explicit_call' := 'do not call this function block directly'}
FUNCTION_BLOCK StaticUniqueDataSetClearTest EXTENDS TOF_Testing.SingleCycleTest
VAR_STAT
	{attribute 'hide'}
	_ClassName : STRING := __POUNAME();
END_VAR
VAR
	_Set : TOF_Collections.UniqueDataSet<7>(valueValidator := 0, valueEqualityComparer := 0);
END_VAR

(*!
<summary>Checks clearing a full inline index and refilling with distinct values.</summary>
*)
METHOD PROTECTED ExecuteTest
VAR
	values : ARRAY [0..6] OF STRING :=
		['String0', 'String1', 'String2', 'String3', 'String4', 'String5', 'String6'];
	i : DINT;
	replacementValues : ARRAY [0..6] OF INT := [11, 12, 13, 14, 15, 16, 17];
END_VAR
FOR i := 6 TO 0 BY -1 DO
	_Set.SetCopy(value := values[i]);
END_FOR

Assert.ThatBool(
	actual := _Set.Full AND_THEN _Set.Length = 7,
	message := "The clear fixture must start full"
).IsTrue();

_Set.Clear();

Assert.ThatBool(
	actual := _Set.Empty AND_THEN _Set.Length = 0 AND_THEN NOT _Set.Full,
	message := "Clearing a full set must make every slot available"
).IsTrue();

Assert.ThatDInt(
	actual := _Set.Capacity,
	message := "Clearing must preserve inline capacity"
).ToBe(expected := DINT#7);

FOR i := 0 TO 6 DO
	Assert.ThatBool(
		actual := _Set.Contains(value := values[i]),
		message := TOF_Core.WideStrings.Concat255("Clear must hide the old value at offset ", TO_WSTRING(i))
	).IsFalse();
END_FOR

FOR i := 0 TO 6 DO
	_Set.SetCopy(value := replacementValues[i]);
END_FOR

Assert.ThatBool(
	actual := _Set.Full AND_THEN _Set.Length = 7,
	message := "Refilling must reuse all seven slots"
).IsTrue();

FOR i := 0 TO 6 DO
	Assert.ThatBool(
		actual := _Set.Contains(value := replacementValues[i]),
		message := TOF_Core.WideStrings.Concat255("Refill must index value ", TO_WSTRING(replacementValues[i]))
	).IsTrue();
END_FOR
END_METHOD

(*!
<summary>Clears the fixture before the runner publishes the result.</summary>
<description>
Also runs after an unexpected exception interrupts the case.
</description>
*)
METHOD PROTECTED AfterTest
_Set.Clear();
END_METHOD

//! <summary>Borrows the concrete class name. Callers must not modify it.</summary>
{attribute 'monitoring' := 'call'}
PROPERTY ClassName : REFERENCE TO STRING
GET
ClassName REF= _ClassName;
END_GET
END_PROPERTY

//! <summary>Borrows the compiler-initialized namespace name. Callers must not modify it.</summary>
{attribute 'monitoring' := 'call'}
PROPERTY NamespaceName : REFERENCE TO STRING
GET
NamespaceName REF= CurrentNamespace.Name;
END_GET
END_PROPERTY

//! <summary>Reports the concrete instance size in bytes.</summary>
{attribute 'monitoring' := 'call'}
PROPERTY SelfSize : ULINT
GET
SelfSize := XSIZEOF(THIS^);
END_GET
END_PROPERTY

END_FUNCTION_BLOCK

// ---- Tests/Collections/Static/StaticUniqueDataSetOverflowTest.TcPOU
(*
SPDX-FileCopyrightText: c 2026 Oleksandr Tiutyk <trofimich@gmail.com>
SPDX-License-Identifier: MIT
License: https://opensource.org/license/mit
*)

(*!
<summary>Checks rejection of a new value at capacity and reuse after removal.</summary>
<description>
Owns a fixed-capacity set and copied values at a stable address. Run from one task.
Teardown clears surviving entries before publication.
</description>
*)

{attribute 'no_assign'}
{attribute 'no_explicit_call' := 'do not call this function block directly'}
FUNCTION_BLOCK StaticUniqueDataSetOverflowTest EXTENDS TOF_Testing.SingleCycleTest
VAR_STAT
	{attribute 'hide'}
	_ClassName : STRING := __POUNAME();
END_VAR
VAR
	_Set : TOF_Collections.UniqueDataSet<7>(valueValidator := 0, valueEqualityComparer := 0);
END_VAR

(*!
<summary>Checks rejection of a new value at capacity and reuse after removal.</summary>
*)
METHOD PROTECTED ExecuteTest
VAR
	values : ARRAY [1..8] OF INT := [1, 2, 3, 4, 5, 6, 7, 8];
	i : DINT;
	removed : BOOL;

	exceptionCode : __SYSTEM.ExceptionCode;
	caught : TOF_Core.IException;
	fullException : TOF_Core.IStaticCollectionFullException;
END_VAR
FOR i := 1 TO 7 DO
	_Set.SetCopy(value := values[i]);
END_FOR

Assert.ThatBool(
	actual := _Set.Full AND_THEN _Set.Length = 7,
	message := "The overflow fixture must start full"
).IsTrue();

__TRY
	_Set.SetCopy(value := values[8]);
__CATCH(exceptionCode)
	caught := TOF_Core.ExceptionManager.GetLastException(
		exceptionCode := exceptionCode,
		catchPointNamespaceName := NamespaceName,
		catchPointPOUName := __POUNAME(),
		catchPointPosition := __POSITION()
	);
__ENDTRY

Assert.ThatBool(
	actual := __QUERYINTERFACE(caught, fullException),
	message := "Adding a new value at capacity must raise StaticCollectionFullException"
).IsTrue();

Assert.ThatBool(
	actual := _Set.Full AND_THEN _Set.Length = 7 AND_THEN _Set.Capacity = 7,
	message := "Rejected insertion must preserve full length and capacity"
).IsTrue();

Assert.ThatBool(
	actual := _Set.Contains(value := values[8]),
	message := "The rejected value must remain absent"
).IsFalse();

FOR i := 1 TO 7 DO
	Assert.ThatBool(
		actual := _Set.Contains(value := values[i]),
		message := TOF_Core.WideStrings.Concat255("Overflow must preserve member ", TO_WSTRING(i))
	).IsTrue();
END_FOR

_Set.TryRemove(value := values[3], removed => removed);

Assert.ThatBool(
	actual := removed,
	message := "Removing a stored member must free a slot"
).IsTrue();

_Set.SetCopy(value := values[8]);

Assert.ThatBool(
	actual := _Set.Full AND_THEN _Set.Length = 7 AND_THEN _Set.Contains(value := values[8]),
	message := "Reusing a slot must make the new member visible"
).IsTrue();

Assert.ThatBool(
	actual := _Set.Contains(value := values[3]),
	message := "Reusing the slot must keep the removed member absent"
).IsFalse();
END_METHOD

(*!
<summary>Clears the fixture before the runner publishes the result.</summary>
<description>
Also runs after an unexpected exception interrupts the case.
</description>
*)
METHOD PROTECTED AfterTest
_Set.Clear();
END_METHOD

//! <summary>Borrows the concrete class name. Callers must not modify it.</summary>
{attribute 'monitoring' := 'call'}
PROPERTY ClassName : REFERENCE TO STRING
GET
ClassName REF= _ClassName;
END_GET
END_PROPERTY

//! <summary>Borrows the compiler-initialized namespace name. Callers must not modify it.</summary>
{attribute 'monitoring' := 'call'}
PROPERTY NamespaceName : REFERENCE TO STRING
GET
NamespaceName REF= CurrentNamespace.Name;
END_GET
END_PROPERTY

//! <summary>Reports the concrete instance size in bytes.</summary>
{attribute 'monitoring' := 'call'}
PROPERTY SelfSize : ULINT
GET
SelfSize := XSIZEOF(THIS^);
END_GET
END_PROPERTY

END_FUNCTION_BLOCK

// ---- Tests/Collections/Dynamic/DynamicListTestGroup.TcPOU
(*
SPDX-FileCopyrightText: c 2026 Oleksandr Tiutyk <trofimich@gmail.com>
SPDX-License-Identifier: MIT
License: https://opensource.org/license/mit
*)

(*!
<summary>Groups dynamic list copying, borrowing, editing, search, sorting and clear cases.</summary>
<description>
Owns the cases, their fixed registration array and any fixtures borrowed by the cases.
Each borrowed fixture is reserved for its case throughout the group lifetime. Use from one task at a stable address.
</description>
*)

{attribute 'no_assign'}
{attribute 'no_explicit_call' := 'do not call this function block directly'}
FUNCTION_BLOCK DynamicListTestGroup EXTENDS TOF_Testing.TestGroup<15>
VAR_STAT
	{attribute 'hide'}
	_ClassName : STRING := __POUNAME();
END_VAR
VAR
	_AppendList : TOF_Collections.List<0>(valueValidator := 0);
	_InsertList : TOF_Collections.List<0>(valueValidator := 0);
	_GetAndSetList : TOF_Collections.List<0>(valueValidator := 0);
	_FindList : TOF_Collections.List<0>(valueValidator := 0);
	_ContainsList : TOF_Collections.List<0>(valueValidator := 0);
	_ContainsGenericList : TOF_Collections.List<0>(valueValidator := 0);
	_RemoveFirstList : TOF_Collections.List<0>(valueValidator := 0);
	_RemoveMatchedList : TOF_Collections.List<0>(valueValidator := 0);
	_RemoveAtList : TOF_Collections.List<0>(valueValidator := 0);
	_SwapList : TOF_Collections.List<0>(valueValidator := 0);
	_AppendGenericList : TOF_Collections.List<0>(valueValidator := 0);
	_InsertGenericList : TOF_Collections.List<0>(valueValidator := 0);
	_GetAndSetGenericList : TOF_Collections.List<0>(valueValidator := 0);

	_Append : ListAppendTest(name := "Append", parent := THIS^, list := _AppendList);
	_Insert : ListInsertTest(name := "Insert", parent := THIS^, list := _InsertList);
	_GetAndSet : ListGetAndSetTest(name := "GetAndSet", parent := THIS^, list := _GetAndSetList);
	_Find : ListFindTest(name := "Find", parent := THIS^, list := _FindList);
	_Contains : ListContainsTest(name := "Contains", parent := THIS^, list := _ContainsList);
	_ContainsGeneric : ListContainsGenericTest(name := "ContainsGeneric", parent := THIS^, list := _ContainsGenericList);
	_RemoveFirst : ListRemoveFirstTest(name := "RemoveFirst", parent := THIS^, list := _RemoveFirstList);
	_RemoveMatched : ListRemoveMatchedTest(name := "RemoveMatched", parent := THIS^, list := _RemoveMatchedList);
	_RemoveAt : ListRemoveAtTest(name := "RemoveAt", parent := THIS^, list := _RemoveAtList);
	_Swap : ListSwapTest(name := "Swap", parent := THIS^, list := _SwapList);
	_Sort : DynamicListSortTest(name := "Sort", parent := THIS^);
	_AppendGeneric : ListAppendGenericTest(name := "AppendGeneric", parent := THIS^, list := _AppendGenericList);
	_InsertGeneric : ListInsertGenericTest(name := "InsertGeneric", parent := THIS^, list := _InsertGenericList);
	_GetAndSetGeneric : ListGetAndSetGenericTest(
		name := "GetAndSetGeneric",
		parent := THIS^,
		list := _GetAndSetGenericList
	);
	_Clear : DynamicListClearTest(name := "Clear", parent := THIS^);

	_Children : ARRAY [0.._ChildCount - 1] OF TOF_Testing.ITestElement :=
	[
		_Append,
		_Insert,
		_GetAndSet,
		_Find,
		_Contains,
		_ContainsGeneric,
		_RemoveFirst,
		_RemoveMatched,
		_RemoveAt,
		_Swap,
		_Sort,
		_AppendGeneric,
		_InsertGeneric,
		_GetAndSetGeneric,
		_Clear
	];
END_VAR

//! <summary>Borrows the fixed child array. Callers must not modify it.</summary>
{attribute 'monitoring' := 'call'}
PROPERTY Children : REFERENCE TO ARRAY [0.._ChildCount - 1] OF TOF_Testing.ITestElement
GET
Children REF= _Children;
END_GET
END_PROPERTY

//! <summary>Borrows the concrete class name. Callers must not modify it.</summary>
{attribute 'monitoring' := 'call'}
PROPERTY ClassName : REFERENCE TO STRING
GET
ClassName REF= _ClassName;
END_GET
END_PROPERTY

//! <summary>Borrows the compiler-initialized namespace name. Callers must not modify it.</summary>
{attribute 'monitoring' := 'call'}
PROPERTY NamespaceName : REFERENCE TO STRING
GET
NamespaceName REF= CurrentNamespace.Name;
END_GET
END_PROPERTY

//! <summary>Reports the concrete instance size in bytes.</summary>
{attribute 'monitoring' := 'call'}
PROPERTY SelfSize : ULINT
GET
SelfSize := XSIZEOF(THIS^);
END_GET
END_PROPERTY

END_FUNCTION_BLOCK

// ---- Tests/Collections/ListAppendTest.TcPOU
(*
SPDX-FileCopyrightText: c 2026 Oleksandr Tiutyk <trofimich@gmail.com>
SPDX-License-Identifier: MIT
License: https://opensource.org/license/mit
*)

(*!
<summary>Checks copy append order and independence from the source.</summary>
<description>
Borrows a group-owned list reserved for this case. Use from one task at a stable address.
Teardown clears the list before publication.
</description>
*)

{attribute 'no_assign'}
{attribute 'no_explicit_call' := 'do not call this function block directly'}
FUNCTION_BLOCK ListAppendTest EXTENDS TOF_Testing.SingleCycleTest
VAR_STAT
	{attribute 'hide'}
	_ClassName : STRING := __POUNAME();
END_VAR
VAR
	_List : TOF_Collections.IList;
END_VAR

(*!
<summary>Binds the list fixture for this case.</summary>
<description>
Stores a borrowed interface without invoking the fixture. The owning group keeps it alive and
reserves it for this case. TestElement initializes the name and parent.
</description>
<param name="name">Display name of this case.</param>
<param name="parent">Group that owns this case.</param>
<param name="list">Required live list reserved for this case.</param>
*)
METHOD FB_init : BOOL
VAR_INPUT
	bInitRetains: BOOL; // TRUE: the retain variables are initialized (reset warm / reset cold)
	bInCopyCode: BOOL; // TRUE: the instance will be copied to the copy code afterward (online change)
	name : WSTRING;
	parent : TOF_Testing.ITestElement;
	list : TOF_Collections.IList;
END_VAR
_List := list;
FB_init := TRUE;
END_METHOD

(*!
<summary>Checks copy append order and independence from the source.</summary>
*)
METHOD PROTECTED ExecuteTest
VAR
	values : ARRAY [0..5] OF STRING := ['String0', 'String1', 'String2', 'String3', 'String4', 'String5'];
	expected : ARRAY [0..2] OF STRING := ['String0', 'String1', 'String2'];
	i : DINT;
END_VAR
_List.AppendCopy(value := values[0]);
_List.AppendCopy(value := values[1]);
_List.AppendCopy(value := values[2]);

values[2] := 'Changed';

Assert.ThatDInt(
	actual := _List.Length,
	message := "Unexpected sequence after Append length"
).ToBe(expected := DINT#3);

FOR i := 0 TO 2 DO
	Assert.ThatString(
		actual := _List.Get(index := i).AsString255(),
		message := TOF_Core.WideStrings.Concat255("Unexpected sequence after Append at index ", TO_WSTRING(i))
	).ToBe(expected := expected[i]);
END_FOR
END_METHOD

(*!
<summary>Clears the fixture before the runner publishes the result.</summary>
<description>
Also runs after an unexpected exception interrupts the case.
</description>
*)
METHOD PROTECTED AfterTest
_List.Clear();
END_METHOD

//! <summary>Borrows the concrete class name. Callers must not modify it.</summary>
{attribute 'monitoring' := 'call'}
PROPERTY ClassName : REFERENCE TO STRING
GET
ClassName REF= _ClassName;
END_GET
END_PROPERTY

//! <summary>Borrows the compiler-initialized namespace name. Callers must not modify it.</summary>
{attribute 'monitoring' := 'call'}
PROPERTY NamespaceName : REFERENCE TO STRING
GET
NamespaceName REF= CurrentNamespace.Name;
END_GET
END_PROPERTY

//! <summary>Reports the concrete instance size in bytes.</summary>
{attribute 'monitoring' := 'call'}
PROPERTY SelfSize : ULINT
GET
SelfSize := XSIZEOF(THIS^);
END_GET
END_PROPERTY

END_FUNCTION_BLOCK

// ---- Tests/Collections/ListInsertTest.TcPOU
(*
SPDX-FileCopyrightText: c 2026 Oleksandr Tiutyk <trofimich@gmail.com>
SPDX-License-Identifier: MIT
License: https://opensource.org/license/mit
*)

(*!
<summary>Checks inserting a copied value and shifting the suffix.</summary>
<description>
Borrows a group-owned list reserved for this case. Use from one task at a stable address.
Teardown clears the list before publication.
</description>
*)

{attribute 'no_assign'}
{attribute 'no_explicit_call' := 'do not call this function block directly'}
FUNCTION_BLOCK ListInsertTest EXTENDS TOF_Testing.SingleCycleTest
VAR_STAT
	{attribute 'hide'}
	_ClassName : STRING := __POUNAME();
END_VAR
VAR
	_List : TOF_Collections.IList;
END_VAR

(*!
<summary>Clears the fixture before the runner publishes the result.</summary>
<description>
Also runs after an unexpected exception interrupts the case.
</description>
*)
METHOD PROTECTED AfterTest
_List.Clear();
END_METHOD

//! <summary>Borrows the concrete class name. Callers must not modify it.</summary>
{attribute 'monitoring' := 'call'}
PROPERTY ClassName : REFERENCE TO STRING
GET
ClassName REF= _ClassName;
END_GET
END_PROPERTY

(*!
<summary>Checks inserting a copied value and shifting the suffix.</summary>
*)
METHOD PROTECTED ExecuteTest
VAR
	values : ARRAY [0..5] OF STRING := ['String0', 'String1', 'String2', 'String3', 'String4', 'String5'];
	expected : ARRAY [0..3] OF STRING := ['String0', 'String5', 'String1', 'String2'];
	i : DINT;
END_VAR
_List.AppendCopy(value := values[0]);
_List.AppendCopy(value := values[1]);
_List.AppendCopy(value := values[2]);

_List.InsertCopy(index := 1, value := values[5]);

Assert.ThatDInt(
	actual := _List.Length,
	message := "Unexpected sequence after Insert length"
).ToBe(expected := DINT#4);

FOR i := 0 TO 3 DO
	Assert.ThatString(
		actual := _List.Get(index := i).AsString255(),
		message := TOF_Core.WideStrings.Concat255("Unexpected sequence after Insert at index ", TO_WSTRING(i))
	).ToBe(expected := expected[i]);
END_FOR
END_METHOD

(*!
<summary>Binds the list fixture for this case.</summary>
<description>
Stores a borrowed interface without invoking the fixture. The owning group keeps it alive and
reserves it for this case. TestElement initializes the name and parent.
</description>
<param name="name">Display name of this case.</param>
<param name="parent">Group that owns this case.</param>
<param name="list">Required live list reserved for this case.</param>
*)
METHOD FB_init : BOOL
VAR_INPUT
	bInitRetains: BOOL; // TRUE: the retain variables are initialized (reset warm / reset cold)
	bInCopyCode: BOOL; // TRUE: the instance will be copied to the copy code afterward (online change)
	name : WSTRING;
	parent : TOF_Testing.ITestElement;
	list : TOF_Collections.IList;
END_VAR
_List := list;
FB_init := TRUE;
END_METHOD

//! <summary>Borrows the compiler-initialized namespace name. Callers must not modify it.</summary>
{attribute 'monitoring' := 'call'}
PROPERTY NamespaceName : REFERENCE TO STRING
GET
NamespaceName REF= CurrentNamespace.Name;
END_GET
END_PROPERTY

//! <summary>Reports the concrete instance size in bytes.</summary>
{attribute 'monitoring' := 'call'}
PROPERTY SelfSize : ULINT
GET
SelfSize := XSIZEOF(THIS^);
END_GET
END_PROPERTY

END_FUNCTION_BLOCK

// ---- Tests/Collections/ListGetAndSetTest.TcPOU
(*
SPDX-FileCopyrightText: c 2026 Oleksandr Tiutyk <trofimich@gmail.com>
SPDX-License-Identifier: MIT
License: https://opensource.org/license/mit
*)

(*!
<summary>Checks replacement of a copied value at one index.</summary>
<description>
Borrows a group-owned list reserved for this case. Use from one task at a stable address.
Teardown clears the list before publication.
</description>
*)

{attribute 'no_assign'}
{attribute 'no_explicit_call' := 'do not call this function block directly'}
FUNCTION_BLOCK ListGetAndSetTest EXTENDS TOF_Testing.SingleCycleTest
VAR_STAT
	{attribute 'hide'}
	_ClassName : STRING := __POUNAME();
END_VAR
VAR
	_List : TOF_Collections.IList;
END_VAR

(*!
<summary>Clears the fixture before the runner publishes the result.</summary>
<description>
Also runs after an unexpected exception interrupts the case.
</description>
*)
METHOD PROTECTED AfterTest
_List.Clear();
END_METHOD

//! <summary>Borrows the concrete class name. Callers must not modify it.</summary>
{attribute 'monitoring' := 'call'}
PROPERTY ClassName : REFERENCE TO STRING
GET
ClassName REF= _ClassName;
END_GET
END_PROPERTY

(*!
<summary>Checks replacement of a copied value at one index.</summary>
*)
METHOD PROTECTED ExecuteTest
VAR
	values : ARRAY [0..5] OF STRING := ['String0', 'String1', 'String2', 'String3', 'String4', 'String5'];
	expected : ARRAY [0..2] OF STRING := ['String0', 'String4', 'String2'];
	i : DINT;
END_VAR
_List.AppendCopy(value := values[0]);
_List.AppendCopy(value := values[1]);
_List.AppendCopy(value := values[2]);

_List.SetCopy(index := 1, value := values[4]);
values[4] := 'Changed';

Assert.ThatDInt(
	actual := _List.Length,
	message := "Unexpected sequence after GetAndSet length"
).ToBe(expected := DINT#3);

FOR i := 0 TO 2 DO
	Assert.ThatString(
		actual := _List.Get(index := i).AsString255(),
		message := TOF_Core.WideStrings.Concat255("Unexpected sequence after GetAndSet at index ", TO_WSTRING(i))
	).ToBe(expected := expected[i]);
END_FOR
END_METHOD

(*!
<summary>Binds the list fixture for this case.</summary>
<description>
Stores a borrowed interface without invoking the fixture. The owning group keeps it alive and
reserves it for this case. TestElement initializes the name and parent.
</description>
<param name="name">Display name of this case.</param>
<param name="parent">Group that owns this case.</param>
<param name="list">Required live list reserved for this case.</param>
*)
METHOD FB_init : BOOL
VAR_INPUT
	bInitRetains: BOOL; // TRUE: the retain variables are initialized (reset warm / reset cold)
	bInCopyCode: BOOL; // TRUE: the instance will be copied to the copy code afterward (online change)
	name : WSTRING;
	parent : TOF_Testing.ITestElement;
	list : TOF_Collections.IList;
END_VAR
_List := list;
FB_init := TRUE;
END_METHOD

//! <summary>Borrows the compiler-initialized namespace name. Callers must not modify it.</summary>
{attribute 'monitoring' := 'call'}
PROPERTY NamespaceName : REFERENCE TO STRING
GET
NamespaceName REF= CurrentNamespace.Name;
END_GET
END_PROPERTY

//! <summary>Reports the concrete instance size in bytes.</summary>
{attribute 'monitoring' := 'call'}
PROPERTY SelfSize : ULINT
GET
SelfSize := XSIZEOF(THIS^);
END_GET
END_PROPERTY

END_FUNCTION_BLOCK

// ---- Tests/Collections/ListFindTest.TcPOU
(*
SPDX-FileCopyrightText: c 2026 Oleksandr Tiutyk <trofimich@gmail.com>
SPDX-License-Identifier: MIT
License: https://opensource.org/license/mit
*)

(*!
<summary>Checks predicate matching, skip, reverse traversal and absence.</summary>
<description>
Borrows a group-owned list reserved for this case. Use from one task at a stable address.
Teardown clears the list before publication.
</description>
*)

{attribute 'no_assign'}
{attribute 'no_explicit_call' := 'do not call this function block directly'}
FUNCTION_BLOCK ListFindTest EXTENDS TOF_Testing.SingleCycleTest
VAR_STAT
	{attribute 'hide'}
	_ClassName : STRING := __POUNAME();
END_VAR
VAR
	_List : TOF_Collections.IList;
	_Predicate : ListStringPredicate;
END_VAR

(*!
<summary>Clears the fixture before the runner publishes the result.</summary>
<description>
Also runs after an unexpected exception interrupts the case.
</description>
*)
METHOD PROTECTED AfterTest
_List.Clear();
END_METHOD

//! <summary>Borrows the concrete class name. Callers must not modify it.</summary>
{attribute 'monitoring' := 'call'}
PROPERTY ClassName : REFERENCE TO STRING
GET
ClassName REF= _ClassName;
END_GET
END_PROPERTY

(*!
<summary>Checks predicate matching, skip, reverse traversal and absence.</summary>
*)
METHOD PROTECTED ExecuteTest
VAR
	values : ARRAY [0..5] OF STRING := ['String0', 'String1', 'String2', 'String3', 'String4', 'String5'];
	found : BOOL;
	index : TOF_Core.DINT_INDEX;
	entry : TOF_Core.GENERIC_VALUE;
END_VAR
_List.AppendCopy(value := values[0]);
_List.AppendCopy(value := values[1]);
_List.AppendCopy(value := values[2]);
_List.AppendCopy(value := values[3]);
_List.AppendCopy(value := values[4]);
_List.AppendCopy(value := values[5]);
_List.AppendCopy(value := values[2]);
_List.AppendCopy(value := values[3]);

_Predicate.Expected := 'String2';

found := _List.FindSingle(predicate := _Predicate, skip := 0, index => index, value => entry);

Assert.ThatBool(
	actual := found AND_THEN index = 2 AND_THEN entry.AsString255() = 'String2',
	message := "Find must return the first match and its value"
).IsTrue();

found := _List.FindSingle(predicate := _Predicate, skip := 1, index => index);

Assert.ThatBool(
	actual := found AND_THEN index = 6,
	message := "Skipping one match must return the second match"
).IsTrue();

found := _List.FindSingle(
	predicate := _Predicate,
	searchDirection := TOF_Core.SEARCH_DIRECTION.FROM_END,
	index => index
);

Assert.ThatBool(
	actual := found AND_THEN index = 6,
	message := "Reverse traversal must find the last occurrence first"
).IsTrue();

found := _List.FindSingle(predicate := _Predicate, skip := 2);

Assert.ThatBool(
	actual := found,
	message := "Skipping both matches must report absence"
).IsFalse();

Assert.ThatDInt(
	actual := _List.Length,
	message := "Find must preserve the list length"
).ToBe(expected := DINT#8);
END_METHOD

(*!
<summary>Binds the list fixture for this case.</summary>
<description>
Stores a borrowed interface without invoking the fixture. The owning group keeps it alive and
reserves it for this case. TestElement initializes the name and parent.
</description>
<param name="name">Display name of this case.</param>
<param name="parent">Group that owns this case.</param>
<param name="list">Required live list reserved for this case.</param>
*)
METHOD FB_init : BOOL
VAR_INPUT
	bInitRetains: BOOL; // TRUE: the retain variables are initialized (reset warm / reset cold)
	bInCopyCode: BOOL; // TRUE: the instance will be copied to the copy code afterward (online change)
	name : WSTRING;
	parent : TOF_Testing.ITestElement;
	list : TOF_Collections.IList;
END_VAR
_List := list;
FB_init := TRUE;
END_METHOD

//! <summary>Borrows the compiler-initialized namespace name. Callers must not modify it.</summary>
{attribute 'monitoring' := 'call'}
PROPERTY NamespaceName : REFERENCE TO STRING
GET
NamespaceName REF= CurrentNamespace.Name;
END_GET
END_PROPERTY

//! <summary>Reports the concrete instance size in bytes.</summary>
{attribute 'monitoring' := 'call'}
PROPERTY SelfSize : ULINT
GET
SelfSize := XSIZEOF(THIS^);
END_GET
END_PROPERTY

END_FUNCTION_BLOCK

// ---- Tests/Collections/ListStringPredicate.TcPOU
(*
SPDX-FileCopyrightText: c 2026 Oleksandr Tiutyk <trofimich@gmail.com>
SPDX-License-Identifier: MIT
License: https://opensource.org/license/mit
*)

(*!
<summary>Matches a borrowed STRING against an expected value.</summary>
<description>
Keeps only the expected text. Check reads each candidate synchronously and makes no allocations.
</description>
*)

{attribute 'no_explicit_call' := 'do not call this function block directly'}
FUNCTION_BLOCK ListStringPredicate EXTENDS TOF_Core.Object IMPLEMENTS TOF_Core.IPredicate
VAR_STAT
	{attribute 'hide'}
	_ClassName : STRING := __POUNAME();
END_VAR
VAR_INPUT
	//! <summary>Value matched by the next Check call.</summary>
	Expected : STRING;
END_VAR

(*!
<summary>Compares a live STRING candidate with the expected text.</summary>
<description>
The input is borrowed for this call and its address is discarded on return.
</description>
*)
METHOD Check : BOOL
VAR_INPUT
	valueToCompare : __SYSTEM.AnyType;
END_VAR
VAR
	candidate : TOF_Core.GENERIC_VALUE;
END_VAR
candidate := TOF_Core.GenericValueFactory.FromAnyType(
	value := valueToCompare,
	isObject := FALSE,
	memoryManagementBehavior :=
		TOF_Core.GENERIC_MEMORY_MANAGEMENT_BEHAVIOR.STORE_ORIGINAL_REFERENCE_AND_NOT_OWNS_MEMORY
);

Check := candidate.TypeClass = TOF_Core.GENERIC_TYPE_CLASS.STRING_8
	AND_THEN candidate.AsString255() = Expected;
END_METHOD

//! <summary>Borrows the concrete class name. Callers must not modify it.</summary>
{attribute 'monitoring' := 'call'}
PROPERTY ClassName : REFERENCE TO STRING
GET
ClassName REF= _ClassName;
END_GET
END_PROPERTY

//! <summary>Borrows the compiler-initialized namespace name. Callers must not modify it.</summary>
{attribute 'monitoring' := 'call'}
PROPERTY NamespaceName : REFERENCE TO STRING
GET
NamespaceName REF= CurrentNamespace.Name;
END_GET
END_PROPERTY

//! <summary>Reports the concrete instance size in bytes.</summary>
{attribute 'monitoring' := 'call'}
PROPERTY SelfSize : ULINT
GET
SelfSize := XSIZEOF(THIS^);
END_GET
END_PROPERTY

END_FUNCTION_BLOCK

// ---- Tests/Collections/ListContainsTest.TcPOU
(*
SPDX-FileCopyrightText: c 2026 Oleksandr Tiutyk <trofimich@gmail.com>
SPDX-License-Identifier: MIT
License: https://opensource.org/license/mit
*)

(*!
<summary>Checks raw membership for a present value, a duplicate and an absent value.</summary>
<description>
Borrows a group-owned list reserved for this case. Use from one task at a stable address.
Teardown clears the list before publication.
</description>
*)

{attribute 'no_assign'}
{attribute 'no_explicit_call' := 'do not call this function block directly'}
FUNCTION_BLOCK ListContainsTest EXTENDS TOF_Testing.SingleCycleTest
VAR_STAT
	{attribute 'hide'}
	_ClassName : STRING := __POUNAME();
END_VAR
VAR
	_List : TOF_Collections.IList;
END_VAR

(*!
<summary>Clears the fixture before the runner publishes the result.</summary>
<description>
Also runs after an unexpected exception interrupts the case.
</description>
*)
METHOD PROTECTED AfterTest
_List.Clear();
END_METHOD

//! <summary>Borrows the concrete class name. Callers must not modify it.</summary>
{attribute 'monitoring' := 'call'}
PROPERTY ClassName : REFERENCE TO STRING
GET
ClassName REF= _ClassName;
END_GET
END_PROPERTY

(*!
<summary>Checks raw membership for a present value, a duplicate and an absent value.</summary>
*)
METHOD PROTECTED ExecuteTest
VAR
	values : ARRAY [0..5] OF STRING := ['String0', 'String1', 'String2', 'String3', 'String4', 'String5'];
END_VAR
_List.AppendCopy(value := values[0]);
_List.AppendCopy(value := values[1]);
_List.AppendCopy(value := values[2]);
_List.AppendCopy(value := values[3]);
_List.AppendCopy(value := values[2]);
_List.AppendCopy(value := values[3]);

Assert.ThatBool(
	actual := _List.Contains(value := values[1]),
	message := "Contains must find String1"
).IsTrue();

Assert.ThatBool(
	actual := _List.Contains(value := values[3]),
	message := "Contains must find the duplicated String3"
).IsTrue();

Assert.ThatBool(
	actual := _List.Contains(value := values[5]),
	message := "Contains must reject absent String5"
).IsFalse();

Assert.ThatDInt(
	actual := _List.Length,
	message := "Contains must preserve all entries"
).ToBe(expected := DINT#6);
END_METHOD

(*!
<summary>Binds the list fixture for this case.</summary>
<description>
Stores a borrowed interface without invoking the fixture. The owning group keeps it alive and
reserves it for this case. TestElement initializes the name and parent.
</description>
<param name="name">Display name of this case.</param>
<param name="parent">Group that owns this case.</param>
<param name="list">Required live list reserved for this case.</param>
*)
METHOD FB_init : BOOL
VAR_INPUT
	bInitRetains: BOOL; // TRUE: the retain variables are initialized (reset warm / reset cold)
	bInCopyCode: BOOL; // TRUE: the instance will be copied to the copy code afterward (online change)
	name : WSTRING;
	parent : TOF_Testing.ITestElement;
	list : TOF_Collections.IList;
END_VAR
_List := list;
FB_init := TRUE;
END_METHOD

//! <summary>Borrows the compiler-initialized namespace name. Callers must not modify it.</summary>
{attribute 'monitoring' := 'call'}
PROPERTY NamespaceName : REFERENCE TO STRING
GET
NamespaceName REF= CurrentNamespace.Name;
END_GET
END_PROPERTY

//! <summary>Reports the concrete instance size in bytes.</summary>
{attribute 'monitoring' := 'call'}
PROPERTY SelfSize : ULINT
GET
SelfSize := XSIZEOF(THIS^);
END_GET
END_PROPERTY

END_FUNCTION_BLOCK

// ---- Tests/Collections/ListContainsGenericTest.TcPOU
(*
SPDX-FileCopyrightText: c 2026 Oleksandr Tiutyk <trofimich@gmail.com>
SPDX-License-Identifier: MIT
License: https://opensource.org/license/mit
*)

(*!
<summary>Checks generic membership using borrowed queries.</summary>
<description>
Borrows a group-owned list reserved for this case. Use from one task at a stable address.
Teardown clears the list before publication.
</description>
*)

{attribute 'no_assign'}
{attribute 'no_explicit_call' := 'do not call this function block directly'}
FUNCTION_BLOCK ListContainsGenericTest EXTENDS TOF_Testing.SingleCycleTest
VAR_STAT
	{attribute 'hide'}
	_ClassName : STRING := __POUNAME();
END_VAR
VAR
	_List : TOF_Collections.IList;
END_VAR

(*!
<summary>Clears the fixture before the runner publishes the result.</summary>
<description>
Also runs after an unexpected exception interrupts the case.
</description>
*)
METHOD PROTECTED AfterTest
_List.Clear();
END_METHOD

//! <summary>Borrows the concrete class name. Callers must not modify it.</summary>
{attribute 'monitoring' := 'call'}
PROPERTY ClassName : REFERENCE TO STRING
GET
ClassName REF= _ClassName;
END_GET
END_PROPERTY

(*!
<summary>Checks generic membership using borrowed queries.</summary>
*)
METHOD PROTECTED ExecuteTest
VAR
	values : ARRAY [0..5] OF STRING := ['String0', 'String1', 'String2', 'String3', 'String4', 'String5'];
	entry : TOF_Core.GENERIC_VALUE;
END_VAR
_List.AppendCopy(value := values[0]);
_List.AppendCopy(value := values[1]);
_List.AppendCopy(value := values[2]);
_List.AppendCopy(value := values[3]);
_List.AppendCopy(value := values[2]);
_List.AppendCopy(value := values[3]);

entry := TOF_Core.GenericValueFactory.FromStringReference(value := values[1]);
Assert.ThatBool(
	actual := _List.ContainsGeneric(value := entry, releaseValue := FALSE),
	message := "ContainsGeneric must find String1"
).IsTrue();

entry := TOF_Core.GenericValueFactory.FromStringReference(value := values[3]);
Assert.ThatBool(
	actual := _List.ContainsGeneric(value := entry, releaseValue := FALSE),
	message := "ContainsGeneric must find the duplicated String3"
).IsTrue();

entry := TOF_Core.GenericValueFactory.FromStringReference(value := values[5]);
Assert.ThatBool(
	actual := _List.ContainsGeneric(value := entry, releaseValue := FALSE),
	message := "ContainsGeneric must reject absent String5"
).IsFalse();

Assert.ThatDInt(
	actual := _List.Length,
	message := "ContainsGeneric must preserve all entries"
).ToBe(expected := DINT#6);
END_METHOD

(*!
<summary>Binds the list fixture for this case.</summary>
<description>
Stores a borrowed interface without invoking the fixture. The owning group keeps it alive and
reserves it for this case. TestElement initializes the name and parent.
</description>
<param name="name">Display name of this case.</param>
<param name="parent">Group that owns this case.</param>
<param name="list">Required live list reserved for this case.</param>
*)
METHOD FB_init : BOOL
VAR_INPUT
	bInitRetains: BOOL; // TRUE: the retain variables are initialized (reset warm / reset cold)
	bInCopyCode: BOOL; // TRUE: the instance will be copied to the copy code afterward (online change)
	name : WSTRING;
	parent : TOF_Testing.ITestElement;
	list : TOF_Collections.IList;
END_VAR
_List := list;
FB_init := TRUE;
END_METHOD

//! <summary>Borrows the compiler-initialized namespace name. Callers must not modify it.</summary>
{attribute 'monitoring' := 'call'}
PROPERTY NamespaceName : REFERENCE TO STRING
GET
NamespaceName REF= CurrentNamespace.Name;
END_GET
END_PROPERTY

//! <summary>Reports the concrete instance size in bytes.</summary>
{attribute 'monitoring' := 'call'}
PROPERTY SelfSize : ULINT
GET
SelfSize := XSIZEOF(THIS^);
END_GET
END_PROPERTY

END_FUNCTION_BLOCK

// ---- Tests/Collections/ListRemoveFirstTest.TcPOU
(*
SPDX-FileCopyrightText: c 2026 Oleksandr Tiutyk <trofimich@gmail.com>
SPDX-License-Identifier: MIT
License: https://opensource.org/license/mit
*)

(*!
<summary>Checks that removing by value removes only the first matching occurrence.</summary>
<description>
Borrows a group-owned list reserved for this case. Use from one task at a stable address.
Teardown clears the list before publication.
</description>
*)

{attribute 'no_assign'}
{attribute 'no_explicit_call' := 'do not call this function block directly'}
FUNCTION_BLOCK ListRemoveFirstTest EXTENDS TOF_Testing.SingleCycleTest
VAR_STAT
	{attribute 'hide'}
	_ClassName : STRING := __POUNAME();
END_VAR
VAR
	_List : TOF_Collections.IList;
END_VAR

(*!
<summary>Clears the fixture before the runner publishes the result.</summary>
<description>
Also runs after an unexpected exception interrupts the case.
</description>
*)
METHOD PROTECTED AfterTest
_List.Clear();
END_METHOD

//! <summary>Borrows the concrete class name. Callers must not modify it.</summary>
{attribute 'monitoring' := 'call'}
PROPERTY ClassName : REFERENCE TO STRING
GET
ClassName REF= _ClassName;
END_GET
END_PROPERTY

(*!
<summary>Checks that removing by value removes only the first matching occurrence.</summary>
*)
METHOD PROTECTED ExecuteTest
VAR
	values : ARRAY [0..5] OF STRING := ['String0', 'String1', 'String2', 'String3', 'String4', 'String5'];
	expected : ARRAY [0..4] OF STRING := ['String0', 'String1', 'String3', 'String4', 'String2'];
	i : DINT;
END_VAR
_List.AppendCopy(value := values[0]);
_List.AppendCopy(value := values[1]);
_List.AppendCopy(value := values[2]);
_List.AppendCopy(value := values[3]);
_List.AppendCopy(value := values[4]);
_List.AppendCopy(value := values[2]);

_List.RemoveFirst(value := values[2]);

Assert.ThatDInt(
	actual := _List.Length,
	message := "Unexpected sequence after RemoveFirst length"
).ToBe(expected := DINT#5);

FOR i := 0 TO 4 DO
	Assert.ThatString(
		actual := _List.Get(index := i).AsString255(),
		message := TOF_Core.WideStrings.Concat255("Unexpected sequence after RemoveFirst at index ", TO_WSTRING(i))
	).ToBe(expected := expected[i]);
END_FOR
END_METHOD

(*!
<summary>Binds the list fixture for this case.</summary>
<description>
Stores a borrowed interface without invoking the fixture. The owning group keeps it alive and
reserves it for this case. TestElement initializes the name and parent.
</description>
<param name="name">Display name of this case.</param>
<param name="parent">Group that owns this case.</param>
<param name="list">Required live list reserved for this case.</param>
*)
METHOD FB_init : BOOL
VAR_INPUT
	bInitRetains: BOOL; // TRUE: the retain variables are initialized (reset warm / reset cold)
	bInCopyCode: BOOL; // TRUE: the instance will be copied to the copy code afterward (online change)
	name : WSTRING;
	parent : TOF_Testing.ITestElement;
	list : TOF_Collections.IList;
END_VAR
_List := list;
FB_init := TRUE;
END_METHOD

//! <summary>Borrows the compiler-initialized namespace name. Callers must not modify it.</summary>
{attribute 'monitoring' := 'call'}
PROPERTY NamespaceName : REFERENCE TO STRING
GET
NamespaceName REF= CurrentNamespace.Name;
END_GET
END_PROPERTY

//! <summary>Reports the concrete instance size in bytes.</summary>
{attribute 'monitoring' := 'call'}
PROPERTY SelfSize : ULINT
GET
SelfSize := XSIZEOF(THIS^);
END_GET
END_PROPERTY

END_FUNCTION_BLOCK

// ---- Tests/Collections/ListRemoveMatchedTest.TcPOU
(*
SPDX-FileCopyrightText: c 2026 Oleksandr Tiutyk <trofimich@gmail.com>
SPDX-License-Identifier: MIT
License: https://opensource.org/license/mit
*)

(*!
<summary>Checks removal of all matches while preserving the order of survivors.</summary>
<description>
Borrows a group-owned list reserved for this case. Use from one task at a stable address.
Teardown clears the list before publication.
</description>
*)

{attribute 'no_assign'}
{attribute 'no_explicit_call' := 'do not call this function block directly'}
FUNCTION_BLOCK ListRemoveMatchedTest EXTENDS TOF_Testing.SingleCycleTest
VAR_STAT
	{attribute 'hide'}
	_ClassName : STRING := __POUNAME();
END_VAR
VAR
	_List : TOF_Collections.IList;
	_Predicate : ListStringPredicate;
END_VAR

(*!
<summary>Clears the fixture before the runner publishes the result.</summary>
<description>
Also runs after an unexpected exception interrupts the case.
</description>
*)
METHOD PROTECTED AfterTest
_List.Clear();
END_METHOD

//! <summary>Borrows the concrete class name. Callers must not modify it.</summary>
{attribute 'monitoring' := 'call'}
PROPERTY ClassName : REFERENCE TO STRING
GET
ClassName REF= _ClassName;
END_GET
END_PROPERTY

(*!
<summary>Checks removal of all matches while preserving the order of survivors.</summary>
*)
METHOD PROTECTED ExecuteTest
VAR
	values : ARRAY [0..5] OF STRING := ['String0', 'String1', 'String2', 'String3', 'String4', 'String5'];
	expected : ARRAY [0..5] OF STRING := ['String0', 'String1', 'String3', 'String4', 'String5', 'String3'];
	i : DINT;
END_VAR
_List.AppendCopy(value := values[0]);
_List.AppendCopy(value := values[1]);
_List.AppendCopy(value := values[2]);
_List.AppendCopy(value := values[3]);
_List.AppendCopy(value := values[4]);
_List.AppendCopy(value := values[5]);
_List.AppendCopy(value := values[2]);
_List.AppendCopy(value := values[3]);

_Predicate.Expected := 'String2';
_List.RemoveMatched(predicate := _Predicate);

Assert.ThatDInt(
	actual := _List.Length,
	message := "Unexpected sequence after RemoveMatched length"
).ToBe(expected := DINT#6);

FOR i := 0 TO 5 DO
	Assert.ThatString(
		actual := _List.Get(index := i).AsString255(),
		message := TOF_Core.WideStrings.Concat255("Unexpected sequence after RemoveMatched at index ", TO_WSTRING(i))
	).ToBe(expected := expected[i]);
END_FOR
END_METHOD

(*!
<summary>Binds the list fixture for this case.</summary>
<description>
Stores a borrowed interface without invoking the fixture. The owning group keeps it alive and
reserves it for this case. TestElement initializes the name and parent.
</description>
<param name="name">Display name of this case.</param>
<param name="parent">Group that owns this case.</param>
<param name="list">Required live list reserved for this case.</param>
*)
METHOD FB_init : BOOL
VAR_INPUT
	bInitRetains: BOOL; // TRUE: the retain variables are initialized (reset warm / reset cold)
	bInCopyCode: BOOL; // TRUE: the instance will be copied to the copy code afterward (online change)
	name : WSTRING;
	parent : TOF_Testing.ITestElement;
	list : TOF_Collections.IList;
END_VAR
_List := list;
FB_init := TRUE;
END_METHOD

//! <summary>Borrows the compiler-initialized namespace name. Callers must not modify it.</summary>
{attribute 'monitoring' := 'call'}
PROPERTY NamespaceName : REFERENCE TO STRING
GET
NamespaceName REF= CurrentNamespace.Name;
END_GET
END_PROPERTY

//! <summary>Reports the concrete instance size in bytes.</summary>
{attribute 'monitoring' := 'call'}
PROPERTY SelfSize : ULINT
GET
SelfSize := XSIZEOF(THIS^);
END_GET
END_PROPERTY

END_FUNCTION_BLOCK

// ---- Tests/Collections/ListRemoveAtTest.TcPOU
(*
SPDX-FileCopyrightText: c 2026 Oleksandr Tiutyk <trofimich@gmail.com>
SPDX-License-Identifier: MIT
License: https://opensource.org/license/mit
*)

(*!
<summary>Checks positional removal and compaction of survivors.</summary>
<description>
Borrows a group-owned list reserved for this case. Use from one task at a stable address.
Teardown clears the list before publication.
</description>
*)

{attribute 'no_assign'}
{attribute 'no_explicit_call' := 'do not call this function block directly'}
FUNCTION_BLOCK ListRemoveAtTest EXTENDS TOF_Testing.SingleCycleTest
VAR_STAT
	{attribute 'hide'}
	_ClassName : STRING := __POUNAME();
END_VAR
VAR
	_List : TOF_Collections.IList;
END_VAR

(*!
<summary>Clears the fixture before the runner publishes the result.</summary>
<description>
Also runs after an unexpected exception interrupts the case.
</description>
*)
METHOD PROTECTED AfterTest
_List.Clear();
END_METHOD

//! <summary>Borrows the concrete class name. Callers must not modify it.</summary>
{attribute 'monitoring' := 'call'}
PROPERTY ClassName : REFERENCE TO STRING
GET
ClassName REF= _ClassName;
END_GET
END_PROPERTY

(*!
<summary>Checks positional removal and compaction of survivors.</summary>
*)
METHOD PROTECTED ExecuteTest
VAR
	values : ARRAY [0..5] OF STRING := ['String0', 'String1', 'String2', 'String3', 'String4', 'String5'];
	expected : ARRAY [0..4] OF STRING := ['String0', 'String1', 'String2', 'String4', 'String5'];
	i : DINT;
END_VAR
_List.AppendCopy(value := values[0]);
_List.AppendCopy(value := values[1]);
_List.AppendCopy(value := values[2]);
_List.AppendCopy(value := values[3]);
_List.AppendCopy(value := values[4]);
_List.AppendCopy(value := values[5]);

_List.RemoveAt(index := 3);

Assert.ThatDInt(
	actual := _List.Length,
	message := "Unexpected sequence after RemoveAt length"
).ToBe(expected := DINT#5);

FOR i := 0 TO 4 DO
	Assert.ThatString(
		actual := _List.Get(index := i).AsString255(),
		message := TOF_Core.WideStrings.Concat255("Unexpected sequence after RemoveAt at index ", TO_WSTRING(i))
	).ToBe(expected := expected[i]);
END_FOR
END_METHOD

(*!
<summary>Binds the list fixture for this case.</summary>
<description>
Stores a borrowed interface without invoking the fixture. The owning group keeps it alive and
reserves it for this case. TestElement initializes the name and parent.
</description>
<param name="name">Display name of this case.</param>
<param name="parent">Group that owns this case.</param>
<param name="list">Required live list reserved for this case.</param>
*)
METHOD FB_init : BOOL
VAR_INPUT
	bInitRetains: BOOL; // TRUE: the retain variables are initialized (reset warm / reset cold)
	bInCopyCode: BOOL; // TRUE: the instance will be copied to the copy code afterward (online change)
	name : WSTRING;
	parent : TOF_Testing.ITestElement;
	list : TOF_Collections.IList;
END_VAR
_List := list;
FB_init := TRUE;
END_METHOD

//! <summary>Borrows the compiler-initialized namespace name. Callers must not modify it.</summary>
{attribute 'monitoring' := 'call'}
PROPERTY NamespaceName : REFERENCE TO STRING
GET
NamespaceName REF= CurrentNamespace.Name;
END_GET
END_PROPERTY

//! <summary>Reports the concrete instance size in bytes.</summary>
{attribute 'monitoring' := 'call'}
PROPERTY SelfSize : ULINT
GET
SelfSize := XSIZEOF(THIS^);
END_GET
END_PROPERTY

END_FUNCTION_BLOCK

// ---- Tests/Collections/ListSwapTest.TcPOU
(*
SPDX-FileCopyrightText: c 2026 Oleksandr Tiutyk <trofimich@gmail.com>
SPDX-License-Identifier: MIT
License: https://opensource.org/license/mit
*)

(*!
<summary>Checks both exchanged endpoints and unchanged middle positions.</summary>
<description>
Borrows a group-owned list reserved for this case. Use from one task at a stable address.
Teardown clears the list before publication.
</description>
*)

{attribute 'no_assign'}
{attribute 'no_explicit_call' := 'do not call this function block directly'}
FUNCTION_BLOCK ListSwapTest EXTENDS TOF_Testing.SingleCycleTest
VAR_STAT
	{attribute 'hide'}
	_ClassName : STRING := __POUNAME();
END_VAR
VAR
	_List : TOF_Collections.IList;
END_VAR

(*!
<summary>Clears the fixture before the runner publishes the result.</summary>
<description>
Also runs after an unexpected exception interrupts the case.
</description>
*)
METHOD PROTECTED AfterTest
_List.Clear();
END_METHOD

//! <summary>Borrows the concrete class name. Callers must not modify it.</summary>
{attribute 'monitoring' := 'call'}
PROPERTY ClassName : REFERENCE TO STRING
GET
ClassName REF= _ClassName;
END_GET
END_PROPERTY

(*!
<summary>Checks both exchanged endpoints and unchanged middle positions.</summary>
*)
METHOD PROTECTED ExecuteTest
VAR
	values : ARRAY [0..5] OF STRING := ['String0', 'String1', 'String2', 'String3', 'String4', 'String5'];
	expected : ARRAY [0..5] OF STRING := ['String5', 'String1', 'String2', 'String3', 'String4', 'String0'];
	i : DINT;
END_VAR
_List.AppendCopy(value := values[0]);
_List.AppendCopy(value := values[1]);
_List.AppendCopy(value := values[2]);
_List.AppendCopy(value := values[3]);
_List.AppendCopy(value := values[4]);
_List.AppendCopy(value := values[5]);

_List.Swap(index1 := 0, index2 := 5);

Assert.ThatDInt(
	actual := _List.Length,
	message := "Unexpected sequence after Swap length"
).ToBe(expected := DINT#6);

FOR i := 0 TO 5 DO
	Assert.ThatString(
		actual := _List.Get(index := i).AsString255(),
		message := TOF_Core.WideStrings.Concat255("Unexpected sequence after Swap at index ", TO_WSTRING(i))
	).ToBe(expected := expected[i]);
END_FOR
END_METHOD

(*!
<summary>Binds the list fixture for this case.</summary>
<description>
Stores a borrowed interface without invoking the fixture. The owning group keeps it alive and
reserves it for this case. TestElement initializes the name and parent.
</description>
<param name="name">Display name of this case.</param>
<param name="parent">Group that owns this case.</param>
<param name="list">Required live list reserved for this case.</param>
*)
METHOD FB_init : BOOL
VAR_INPUT
	bInitRetains: BOOL; // TRUE: the retain variables are initialized (reset warm / reset cold)
	bInCopyCode: BOOL; // TRUE: the instance will be copied to the copy code afterward (online change)
	name : WSTRING;
	parent : TOF_Testing.ITestElement;
	list : TOF_Collections.IList;
END_VAR
_List := list;
FB_init := TRUE;
END_METHOD

//! <summary>Borrows the compiler-initialized namespace name. Callers must not modify it.</summary>
{attribute 'monitoring' := 'call'}
PROPERTY NamespaceName : REFERENCE TO STRING
GET
NamespaceName REF= CurrentNamespace.Name;
END_GET
END_PROPERTY

//! <summary>Reports the concrete instance size in bytes.</summary>
{attribute 'monitoring' := 'call'}
PROPERTY SelfSize : ULINT
GET
SelfSize := XSIZEOF(THIS^);
END_GET
END_PROPERTY

END_FUNCTION_BLOCK

// ---- Tests/Collections/Dynamic/DynamicListSortTest.TcPOU
(*
SPDX-FileCopyrightText: c 2026 Oleksandr Tiutyk <trofimich@gmail.com>
SPDX-License-Identifier: MIT
License: https://opensource.org/license/mit
*)

(*!
<summary>Checks both sort directions for small strings and large DINT input.</summary>
<description>
Owns a list and its copied entries. Use from one task at a stable address.
Teardown clears surviving entries before publication.
</description>
*)

{attribute 'no_assign'}
{attribute 'no_explicit_call' := 'do not call this function block directly'}
FUNCTION_BLOCK DynamicListSortTest EXTENDS TOF_Testing.SingleCycleTest
VAR_STAT
	{attribute 'hide'}
	_ClassName : STRING := __POUNAME();
END_VAR
VAR
	_List : TOF_Collections.List<0>(valueValidator := 0);
END_VAR

(*!
<summary>Checks both sort directions for small strings and large DINT input.</summary>
*)
METHOD PROTECTED ExecuteTest
VAR
	text : ARRAY [0..15] OF STRING := [
		'S00', 'S01', 'S02', 'S03', 'S04', 'S05', 'S06', 'S07',
		'S08', 'S09', 'S10', 'S11', 'S12', 'S13', 'S14', 'S15'
	];
	i : DINT;
	value : DINT;
END_VAR
FOR i := 0 TO 15 DO
	_List.AppendCopy(value := text[i]);
END_FOR

_List.Sort(
	comparer := TOF_Comparison.StandardComparers.StringComparer,
	direction := TOF_Core.SORT_DIRECTION.DESCENDING
);

FOR i := 0 TO 15 DO
	Assert.ThatString(
		actual := _List.Get(index := i).AsString255(),
		message := TOF_Core.WideStrings.Concat255("DESCENDING STRING sort at index ", TO_WSTRING(i))
	).ToBe(expected := text[15 - i]);
END_FOR

_List.Sort(
	comparer := TOF_Comparison.StandardComparers.StringComparer,
	direction := TOF_Core.SORT_DIRECTION.ASCENDING
);

FOR i := 0 TO 15 DO
	Assert.ThatString(
		actual := _List.Get(index := i).AsString255(),
		message := TOF_Core.WideStrings.Concat255("ASCENDING STRING sort at index ", TO_WSTRING(i))
	).ToBe(expected := text[i]);
END_FOR

_List.Clear();

FOR i := 0 TO 100 DO
	value := i;
	_List.AppendCopy(value := value);
END_FOR

_List.Sort(
	comparer := TOF_Comparison.StandardComparers.DIntComparer,
	direction := TOF_Core.SORT_DIRECTION.DESCENDING
);

FOR i := 0 TO 100 DO
	Assert.ThatDInt(
		actual := _List.Get(index := i).AsDInt(),
		message := TOF_Core.WideStrings.Concat255("DESCENDING DINT sort at index ", TO_WSTRING(i))
	).ToBe(expected := 100 - i);
END_FOR

_List.Sort(
	comparer := TOF_Comparison.StandardComparers.DIntComparer,
	direction := TOF_Core.SORT_DIRECTION.ASCENDING
);

FOR i := 0 TO 100 DO
	Assert.ThatDInt(
		actual := _List.Get(index := i).AsDInt(),
		message := TOF_Core.WideStrings.Concat255("ASCENDING DINT sort at index ", TO_WSTRING(i))
	).ToBe(expected := i);
END_FOR
END_METHOD

(*!
<summary>Clears the fixture before the runner publishes the result.</summary>
<description>
Also runs after an unexpected exception interrupts the case.
</description>
*)
METHOD PROTECTED AfterTest
_List.Clear();
END_METHOD

//! <summary>Borrows the concrete class name. Callers must not modify it.</summary>
{attribute 'monitoring' := 'call'}
PROPERTY ClassName : REFERENCE TO STRING
GET
ClassName REF= _ClassName;
END_GET
END_PROPERTY

//! <summary>Borrows the compiler-initialized namespace name. Callers must not modify it.</summary>
{attribute 'monitoring' := 'call'}
PROPERTY NamespaceName : REFERENCE TO STRING
GET
NamespaceName REF= CurrentNamespace.Name;
END_GET
END_PROPERTY

//! <summary>Reports the concrete instance size in bytes.</summary>
{attribute 'monitoring' := 'call'}
PROPERTY SelfSize : ULINT
GET
SelfSize := XSIZEOF(THIS^);
END_GET
END_PROPERTY

END_FUNCTION_BLOCK

// ---- Tests/Collections/ListAppendGenericTest.TcPOU
(*
SPDX-FileCopyrightText: c 2026 Oleksandr Tiutyk <trofimich@gmail.com>
SPDX-License-Identifier: MIT
License: https://opensource.org/license/mit
*)

(*!
<summary>Checks appending borrowed strings without cloning or adopting them.</summary>
<description>
Borrows a group-owned list reserved for this case. Use from one task at a stable address.
Teardown clears the list before publication.
</description>
*)

